LIN {X 0,Y 672.032,Z 834.911,A -85,B 0,C 180,E1 31418.47,E2 31418.47} C_VEL
LIN {X 0,Y 671.95,Z 841.394,A -85,B 0,C 180,E1 31416.751,E2 31416.751} C_VEL
LIN {X 0,Y 671.913,Z 846.943,A -85,B 0,C 180,E1 31414.78,E2 31414.78} C_VEL
LIN {X 0,Y 671.901,Z 850.246,A -85,B 0,C 180,E1 31412.986,E2 31412.986} C_VEL
LIN {X 0,Y 671.897,Z 851.95,A -85,B 0,C 180,E1 31411.364,E2 31411.364} C_VEL
LIN {X 0,Y 671.9,Z 852.431,A -85,B 0,C 180,E1 31409.574,E2 31409.574} C_VEL
LIN {X 0,Y 671.909,Z 851.064,A -85,B 0,C 180,E1 31407.527,E2 31407.527} C_VEL
LIN {X 0,Y 671.923,Z 848.206,A -85,B 0,C 180,E1 31405.733,E2 31405.733} C_VEL
LIN {X 0,Y 671.94,Z 844.025,A -85,B 0,C 180,E1 31404.021,E2 31404.021} C_VEL
LIN {X 0,Y 671.981,Z 838.375,A -85,B 0,C 180,E1 31402.304,E2 31402.304} C_VEL
LIN {X 0,Y 672.106,Z 829.893,A -85,B 0,C 180,E1 31400.322,E2 31400.322} C_VEL
LIN {X 0,Y 672.271,Z 821.072,A -85,B 0,C 180,E1 31398.678,E2 31398.678} C_VEL
LIN {X 0,Y 672.494,Z 811.756,A -85,B 0,C 180,E1 31397.201,E2 31397.201} C_VEL
LIN {X 0,Y 672.852,Z 799.566,A -85,B 0,C 180,E1 31395.543,E2 31395.543} C_VEL
LIN {X 0,Y 673.329,Z 784.965,A -85,B 0,C 180,E1 31393.877,E2 31393.877} C_VEL
LIN {X 0,Y 673.81,Z 771.549,A -85,B 0,C 180,E1 31392.557,E2 31392.557} C_VEL
LIN {X 0,Y 674.343,Z 757.55,A -85,B 0,C 180,E1 31391.35,E2 31391.35} C_VEL
LIN {X 0,Y 674.979,Z 741.859,A -85,B 0,C 180,E1 31390.165,E2 31390.165} C_VEL
LIN {X 0,Y 675.763,Z 721.934,A -85,B 0,C 180,E1 31388.882,E2 31388.882} C_VEL
LIN {X 0,Y 676.425,Z 704.738,A -85,B 0,C 180,E1 31387.947,E2 31387.947} C_VEL
LIN {X 0,Y 676.991,Z 688.587,A -85,B 0,C 180,E1 31387.188,E2 31387.188} C_VEL
LIN {X 0,Y 677.555,Z 671.856,A -85,B 0,C 180,E1 31386.519,E2 31386.519} C_VEL
LIN {X 0,Y 678.053,Z 655.221,A -85,B 0,C 180,E1 31385.96,E2 31385.96} C_VEL
LIN {X 0,Y 678.51,Z 638.285,A -85,B 0,C 180,E1 31385.494,E2 31385.494} C_VEL
LIN {X 0,Y 678.88,Z 621.075,A -85,B 0,C 180,E1 31385.12,E2 31385.12} C_VEL
LIN {X 0,Y 679.16,Z 603.568,A -85,B 0,C 180,E1 31384.84,E2 31384.84} C_VEL
LIN {X 0,Y 681.182,Z 326.681,A -85,B 0,C 180,E1 31381.687,E2 31381.687} C_VEL
LIN {X 0,Y 681.006,Z 317.975,A -85,B 0,C 180,E1 31381.575,E2 31381.575} C_VEL
LIN {X 0,Y 679.405,Z 309.493,A -85,B 0,C 180,E1 31381.377,E2 31381.377} C_VEL
LIN {X 0,Y 680.471,Z 276.701,A -85,B 0,C 180,E1 31379.001,E2 31379.001} C_VEL
LIN {X 0,Y 681.79,Z 234.937,A -85,B 0,C 180,E1 31375.957,E2 31375.957} C_VEL
LIN {X 0,Y 681.872,Z 225.908,A -85,B 0,C 180,E1 31375.284,E2 31375.284} C_VEL
LIN {X 0,Y 675.939,Z 210.334,A -85,B 0,C 180,E1 31373.798,E2 31373.798} C_VEL
LIN {X 0,Y 672.552,Z 201.457,A -85,B 0,C 180,E1 31372.978,E2 31372.978} C_VEL
LIN {X 0,Y 672.581,Z 201.453,A -85,B 0,C 180,E1 31370.042,E2 31370.042} C_VEL
LIN {X 0,Y 672.558,Z 201.452,A -85,B 0,C 180,E1 31367.085,E2 31367.085} C_VEL
LIN {X 0,Y 672.581,Z 201.448,A -85,B 0,C 180,E1 31364.087,E2 31364.087} C_VEL
LIN {X 0,Y 672.561,Z 201.45,A -85,B 0,C 180,E1 31361.081,E2 31361.081} C_VEL
LIN {X 0,Y 672.58,Z 201.45,A -85,B 0,C 180,E1 31358.095,E2 31358.095} C_VEL
LIN {X 0,Y 672.565,Z 201.448,A -85,B 0,C 180,E1 31355.02,E2 31355.02} C_VEL
LIN {X 0,Y 672.578,Z 201.451,A -85,B 0,C 180,E1 31352.055,E2 31352.055} C_VEL
LIN {X 0,Y 672.57,Z 201.443,A -85,B 0,C 180,E1 31349.054,E2 31349.054} C_VEL
LIN {X 0,Y 672.575,Z 201.452,A -85,B 0,C 180,E1 31346.013,E2 31346.013} C_VEL
LIN {X 0,Y 672.573,Z 201.435,A -85,B 0,C 180,E1 31343.016,E2 31343.016} C_VEL
LIN {X 0,Y 672.572,Z 201.448,A -85,B 0,C 180,E1 31339.995,E2 31339.995} C_VEL
LIN {X 0,Y 672.574,Z 201.438,A -85,B 0,C 180,E1 31336.941,E2 31336.941} C_VEL
LIN {X 0,Y 672.569,Z 201.445,A -85,B 0,C 180,E1 31333.936,E2 31333.936} C_VEL
LIN {X 0,Y 672.576,Z 201.439,A -85,B 0,C 180,E1 31330.883,E2 31330.883} C_VEL
LIN {X 0,Y 672.565,Z 201.446,A -85,B 0,C 180,E1 31327.861,E2 31327.861} C_VEL
LIN {X 0,Y 672.579,Z 201.437,A -85,B 0,C 180,E1 31324.861,E2 31324.861} C_VEL
LIN {X 0,Y 672.561,Z 201.448,A -85,B 0,C 180,E1 31321.789,E2 31321.789} C_VEL
LIN {X 0,Y 672.581,Z 201.432,A -85,B 0,C 180,E1 31318.807,E2 31318.807} C_VEL
LIN {X 0,Y 672.557,Z 201.451,A -85,B 0,C 180,E1 31315.737,E2 31315.737} C_VEL
LIN {X 0,Y 672.582,Z 201.433,A -85,B 0,C 180,E1 31312.74,E2 31312.74} C_VEL
LIN {X 0,Y 672.555,Z 201.452,A -85,B 0,C 180,E1 31309.723,E2 31309.723} C_VEL
LIN {X 0,Y 672.586,Z 201.445,A -85,B 0,C 180,E1 31306.765,E2 31306.765} C_VEL
LIN {X 0,Y 672.554,Z 201.454,A -85,B 0,C 180,E1 31303.77,E2 31303.77} C_VEL
LIN {X 0,Y 672.582,Z 201.444,A -85,B 0,C 180,E1 31300.819,E2 31300.819} C_VEL
LIN {X 0,Y 672.552,Z 201.454,A -85,B 0,C 180,E1 31297.721,E2 31297.721} C_VEL
LIN {X 0,Y 672.581,Z 201.446,A -85,B 0,C 180,E1 31294.744,E2 31294.744} C_VEL
LIN {X 0,Y 672.547,Z 201.453,A -85,B 0,C 180,E1 31291.659,E2 31291.659} C_VEL
LIN {X 0,Y 672.578,Z 201.447,A -85,B 0,C 180,E1 31288.74,E2 31288.74} C_VEL
LIN {X 0,Y 672.549,Z 201.455,A -85,B 0,C 180,E1 31285.704,E2 31285.704} C_VEL
LIN {X 0,Y 672.559,Z 201.449,A -85,B 0,C 180,E1 31282.832,E2 31282.832} C_VEL
LIN {X 0,Y 672.548,Z 201.456,A -85,B 0,C 180,E1 31279.702,E2 31279.702} C_VEL
LIN {X 0,Y 672.55,Z 201.452,A -85,B 0,C 180,E1 31276.851,E2 31276.851} C_VEL
LIN {X 0,Y 672.552,Z 201.458,A -85,B 0,C 180,E1 31273.735,E2 31273.735} C_VEL
LIN {X 0,Y 672.57,Z 201.682,A -85,B 0,C 180,E1 31272.914,E2 31272.914} C_VEL
LIN {X 0,Y 673.919,Z 205.007,A -85,B 0,C 180,E1 31272.615,E2 31272.615} C_VEL
LIN {X 0,Y 682.61,Z 222.727,A -85,B 0,C 180,E1 31270.965,E2 31270.965} C_VEL
LIN {X 0,Y 686.788,Z 232.051,A -85,B 0,C 180,E1 31270.19,E2 31270.19} C_VEL
LIN {X 0,Y 684.973,Z 290.804,A -85,B 0,C 180,E1 31267.339,E2 31267.339} C_VEL
LIN {X 0,Y 684.73,Z 300.754,A -85,B 0,C 180,E1 31266.874,E2 31266.874} C_VEL
LIN {X 0,Y 686.841,Z 315.173,A -85,B 0,C 180,E1 31266.576,E2 31266.576} C_VEL
LIN {X 0,Y 685.386,Z 510.12,A -85,B 0,C 180,E1 31264.28,E2 31264.28} C_VEL
LIN {X 0,Y 683.704,Z 691.141,A -85,B 0,C 180,E1 31262.122,E2 31262.122} C_VEL
LIN {X 0,Y 683.128,Z 716.495,A -85,B 0,C 180,E1 31261.672,E2 31261.672} C_VEL
LIN {X 0,Y 682.438,Z 738.1,A -85,B 0,C 180,E1 31261.152,E2 31261.152} C_VEL
LIN {X 0,Y 681.652,Z 761.266,A -85,B 0,C 180,E1 31260.451,E2 31260.451} C_VEL
LIN {X 0,Y 680.761,Z 782.216,A -85,B 0,C 180,E1 31259.668,E2 31259.668} C_VEL
LIN {X 0,Y 679.885,Z 802.279,A -85,B 0,C 180,E1 31258.793,E2 31258.793} C_VEL
LIN {X 0,Y 678.731,Z 825.506,A -85,B 0,C 180,E1 31257.601,E2 31257.601} C_VEL
LIN {X 0,Y 677.787,Z 844.732,A -85,B 0,C 180,E1 31256.457,E2 31256.457} C_VEL
LIN {X 0,Y 676.663,Z 866.009,A -85,B 0,C 180,E1 31255,E2 31255} C_VEL
LIN {X 0,Y 675.802,Z 883.401,A -85,B 0,C 180,E1 31253.638,E2 31253.638} C_VEL
LIN {X 0,Y 674.846,Z 902.606,A -85,B 0,C 180,E1 31251.924,E2 31251.924} C_VEL
LIN {X 0,Y 674.159,Z 917.749,A -85,B 0,C 180,E1 31250.386,E2 31250.386} C_VEL
LIN {X 0,Y 673.471,Z 933.816,A -85,B 0,C 180,E1 31248.525,E2 31248.525} C_VEL
LIN {X 0,Y 673.017,Z 946.526,A -85,B 0,C 180,E1 31246.84,E2 31246.84} C_VEL
LIN {X 0,Y 672.589,Z 959.764,A -85,B 0,C 180,E1 31244.815,E2 31244.815} C_VEL
LIN {X 0,Y 672.315,Z 969.606,A -85,B 0,C 180,E1 31243.058,E2 31243.058} C_VEL
LIN {X 0,Y 672.101,Z 979.477,A -85,B 0,C 180,E1 31240.978,E2 31240.978} C_VEL
LIN {X 0,Y 672.004,Z 986.514,A -85,B 0,C 180,E1 31239.161,E2 31239.161} C_VEL
LIN {X 0,Y 671.934,Z 992.507,A -85,B 0,C 180,E1 31237.267,E2 31237.267} C_VEL
LIN {X 0,Y 671.893,Z 997.337,A -85,B 0,C 180,E1 31235.208,E2 31235.208} C_VEL
LIN {X 0,Y 671.908,Z 1000.237,A -85,B 0,C 180,E1 31233.413,E2 31233.413} C_VEL
LIN {X 0,Y 671.908,Z 1002.17,A -85,B 0,C 180,E1 31231.279,E2 31231.279} C_VEL
LIN {X 0,Y 671.882,Z 1002.351,A -85,B 0,C 180,E1 31229.403,E2 31229.403} C_VEL
LIN {X 0,Y 671.907,Z 1001.363,A -85,B 0,C 180,E1 31227.612,E2 31227.612} C_VEL
LIN {X 0,Y 671.918,Z 998.608,A -85,B 0,C 180,E1 31225.476,E2 31225.476} C_VEL
LIN {X 0,Y 671.925,Z 994.689,A -85,B 0,C 180,E1 31223.592,E2 31223.592} C_VEL
LIN {X 0,Y 671.975,Z 989.201,A -85,B 0,C 180,E1 31221.615,E2 31221.615} C_VEL
LIN {X 0,Y 672.091,Z 981.605,A -85,B 0,C 180,E1 31219.543,E2 31219.543} C_VEL
LIN {X 0,Y 672.253,Z 973.118,A -85,B 0,C 180,E1 31217.632,E2 31217.632} C_VEL
LIN {X 0,Y 672.515,Z 962.354,A -85,B 0,C 180,E1 31215.623,E2 31215.623} C_VEL
LIN {X 0,Y 672.843,Z 951.388,A -85,B 0,C 180,E1 31213.865,E2 31213.865} C_VEL
LIN {X 0,Y 673.361,Z 936.945,A -85,B 0,C 180,E1 31211.871,E2 31211.871} C_VEL
LIN {X 0,Y 673.931,Z 922.728,A -85,B 0,C 180,E1 31210.161,E2 31210.161} C_VEL
LIN {X 0,Y 674.685,Z 906.31,A -85,B 0,C 180,E1 31208.436,E2 31208.436} C_VEL
LIN {X 0,Y 675.451,Z 890.139,A -85,B 0,C 180,E1 31206.935,E2 31206.935} C_VEL
LIN {X 0,Y 676.436,Z 870.867,A -85,B 0,C 180,E1 31205.364,E2 31205.364} C_VEL
LIN {X 0,Y 677.326,Z 853.071,A -85,B 0,C 180,E1 31204.09,E2 31204.09} C_VEL
LIN {X 0,Y 678.489,Z 830.879,A -85,B 0,C 180,E1 31202.704,E2 31202.704} C_VEL
LIN {X 0,Y 679.431,Z 811.337,A -85,B 0,C 180,E1 31201.649,E2 31201.649} C_VEL
LIN {X 0,Y 680.53,Z 787.863,A -85,B 0,C 180,E1 31200.562,E2 31200.562} C_VEL
LIN {X 0,Y 681.37,Z 767.685,A -85,B 0,C 180,E1 31199.778,E2 31199.778} C_VEL
LIN {X 0,Y 682.256,Z 745.15,A -85,B 0,C 180,E1 31199.042,E2 31199.042} C_VEL
LIN {X 0,Y 682.957,Z 721.163,A -85,B 0,C 180,E1 31198.429,E2 31198.429} C_VEL
LIN {X 0,Y 683.574,Z 698.388,A -85,B 0,C 180,E1 31197.987,E2 31197.987} C_VEL
LIN {X 0,Y 684.015,Z 664.777,A -85,B 0,C 180,E1 31197.547,E2 31197.547} C_VEL
LIN {X 0,Y 686.084,Z 426.859,A -85,B 0,C 180,E1 31194.728,E2 31194.728} C_VEL
LIN {X 0,Y 686.203,Z 312.509,A -85,B 0,C 180,E1 31193.45,E2 31193.45} C_VEL
LIN {X 0,Y 684.133,Z 300.68,A -85,B 0,C 180,E1 31193.219,E2 31193.219} C_VEL
LIN {X 0,Y 685,Z 265.459,A -85,B 0,C 180,E1 31191.55,E2 31191.55} C_VEL
LIN {X 0,Y 686.519,Z 233.708,A -85,B 0,C 180,E1 31189.927,E2 31189.927} C_VEL
LIN {X 0,Y 686.523,Z 231.357,A -85,B 0,C 180,E1 31189.791,E2 31189.791} C_VEL
LIN {X 0,Y 680.861,Z 218.547,A -85,B 0,C 180,E1 31188.502,E2 31188.502} C_VEL
LIN {X 0,Y 676.932,Z 210.351,A -85,B 0,C 180,E1 31187.483,E2 31187.483} C_VEL
LIN {X 0,Y 674.606,Z 205.849,A -85,B 0,C 180,E1 31186.823,E2 31186.823} C_VEL
LIN {X 0,Y 672.75,Z 202.49,A -85,B 0,C 180,E1 31186.247,E2 31186.247} C_VEL
LIN {X 0,Y 672.552,Z 201.458,A -85,B 0,C 180,E1 31186.094,E2 31186.094} C_VEL
LIN {X 0,Y 672.565,Z 201.456,A -85,B 0,C 180,E1 31182.914,E2 31182.914} C_VEL
LIN {X 0,Y 672.538,Z 201.46,A -85,B 0,C 180,E1 31180.073,E2 31180.073} C_VEL
LIN {X 0,Y 672.614,Z 201.669,A -85,B 0,C 180,E1 31177.633,E2 31177.633} C_VEL
LIN {X 0,Y 674.124,Z 205.273,A -85,B 0,C 180,E1 31177.062,E2 31177.062} C_VEL
LIN {X 0,Y 675.014,Z 206.813,A -85,B 0,C 180,E1 31176.809,E2 31176.809} C_VEL
LIN {X 0,Y 678.723,Z 215.05,A -85,B 0,C 180,E1 31175.689,E2 31175.689} C_VEL
LIN {X 0,Y 683.33,Z 226.73,A -85,B 0,C 180,E1 31174.383,E2 31174.383} C_VEL
LIN {X 0,Y 683.402,Z 229.375,A -85,B 0,C 180,E1 31174.183,E2 31174.183} C_VEL
LIN {X 0,Y 680.701,Z 272.496,A -85,B 0,C 180,E1 31171.412,E2 31171.412} C_VEL
LIN {X 0,Y 678.57,Z 326.363,A -85,B 0,C 180,E1 31168.134,E2 31168.134} C_VEL
LIN {X 0,Y 677.146,Z 378.659,A -85,B 0,C 180,E1 31165.074,E2 31165.074} C_VEL
LIN {X 0,Y 675.934,Z 433.54,A -85,B 0,C 180,E1 31161.951,E2 31161.951} C_VEL
LIN {X 0,Y 675.545,Z 457.444,A -85,B 0,C 180,E1 31160.632,E2 31160.632} C_VEL
LIN {X 0,Y 678.294,Z 481.315,A -85,B 0,C 180,E1 31160.165,E2 31160.165} C_VEL
LIN {X 0,Y 676.325,Z 608.391,A -85,B 0,C 180,E1 31158.536,E2 31158.536} C_VEL
LIN {X 0,Y 675.634,Z 682.185,A -85,B 0,C 180,E1 31157.622,E2 31157.622} C_VEL
LIN {X 0,Y 675.344,Z 701.727,A -85,B 0,C 180,E1 31157.222,E2 31157.222} C_VEL
LIN {X 0,Y 675.02,Z 719.823,A -85,B 0,C 180,E1 31156.7,E2 31156.7} C_VEL
LIN {X 0,Y 674.636,Z 737.26,A -85,B 0,C 180,E1 31156.046,E2 31156.046} C_VEL
LIN {X 0,Y 674.245,Z 754.12,A -85,B 0,C 180,E1 31155.251,E2 31155.251} C_VEL
LIN {X 0,Y 673.837,Z 770.294,A -85,B 0,C 180,E1 31154.31,E2 31154.31} C_VEL
LIN {X 0,Y 673.428,Z 785.113,A -85,B 0,C 180,E1 31153.262,E2 31153.262} C_VEL
LIN {X 0,Y 673.048,Z 798.81,A -85,B 0,C 180,E1 31152.091,E2 31152.091} C_VEL
LIN {X 0,Y 672.736,Z 810.592,A -85,B 0,C 180,E1 31150.881,E2 31150.881} C_VEL
LIN {X 0,Y 672.473,Z 821.059,A -85,B 0,C 180,E1 31149.586,E2 31149.586} C_VEL
LIN {X 0,Y 672.265,Z 830.19,A -85,B 0,C 180,E1 31148.209,E2 31148.209} C_VEL
LIN {X 0,Y 672.124,Z 837.938,A -85,B 0,C 180,E1 31146.749,E2 31146.749} C_VEL
LIN {X 0,Y 672.045,Z 844.23,A -85,B 0,C 180,E1 31145.207,E2 31145.207} C_VEL
LIN {X 0,Y 671.982,Z 848.97,A -85,B 0,C 180,E1 31143.583,E2 31143.583} C_VEL
LIN {X 0,Y 671.955,Z 852.015,A -85,B 0,C 180,E1 31141.876,E2 31141.876} C_VEL
LIN {X 0,Y 671.948,Z 853.148,A -85,B 0,C 180,E1 31140.256,E2 31140.256} C_VEL
LIN {X 0,Y 671.945,Z 852.596,A -85,B 0,C 180,E1 31138.636,E2 31138.636} C_VEL
LIN {X 0,Y 671.96,Z 850.344,A -85,B 0,C 180,E1 31137.015,E2 31137.015} C_VEL
LIN {X 0,Y 671.989,Z 846.324,A -85,B 0,C 180,E1 31135.391,E2 31135.391} C_VEL
LIN {X 0,Y 672.056,Z 840.398,A -85,B 0,C 180,E1 31133.765,E2 31133.765} C_VEL
LIN {X 0,Y 672.168,Z 832.667,A -85,B 0,C 180,E1 31132.187,E2 31132.187} C_VEL
LIN {X 0,Y 672.345,Z 823.743,A -85,B 0,C 180,E1 31130.757,E2 31130.757} C_VEL
LIN {X 0,Y 672.591,Z 813.122,A -85,B 0,C 180,E1 31129.377,E2 31129.377} C_VEL
LIN {X 0,Y 672.898,Z 800.975,A -85,B 0,C 180,E1 31128.08,E2 31128.08} C_VEL
LIN {X 0,Y 673.268,Z 787.237,A -85,B 0,C 180,E1 31126.866,E2 31126.866} C_VEL
LIN {X 0,Y 673.678,Z 772.328,A -85,B 0,C 180,E1 31125.776,E2 31125.776} C_VEL
LIN {X 0,Y 674.102,Z 756.538,A -85,B 0,C 180,E1 31124.823,E2 31124.823} C_VEL
LIN {X 0,Y 674.498,Z 739.713,A -85,B 0,C 180,E1 31123.994,E2 31123.994} C_VEL
LIN {X 0,Y 674.919,Z 721.886,A -85,B 0,C 180,E1 31123.297,E2 31123.297} C_VEL
LIN {X 0,Y 675.274,Z 702.619,A -85,B 0,C 180,E1 31122.724,E2 31122.724} C_VEL
LIN {X 0,Y 675.562,Z 683.284,A -85,B 0,C 180,E1 31122.32,E2 31122.32} C_VEL
LIN {X 0,Y 675.824,Z 651.623,A -85,B 0,C 180,E1 31121.921,E2 31121.921} C_VEL
LIN {X 0,Y 676.454,Z 561.656,A -85,B 0,C 180,E1 31120.895,E2 31120.895} C_VEL
LIN {X 0,Y 675.607,Z 554.064,A -85,B 0,C 180,E1 31120.777,E2 31120.777} C_VEL
LIN {X 0,Y 669.963,Z 534.195,A -85,B 0,C 180,E1 31120.351,E2 31120.351} C_VEL
LIN {X 0,Y 669.337,Z 527.67,A -85,B 0,C 180,E1 31120.25,E2 31120.25} C_VEL
LIN {X 0,Y 669.559,Z 478.594,A -85,B 0,C 180,E1 31119.656,E2 31119.656} C_VEL
LIN {X 0,Y 667.897,Z 464.609,A -85,B 0,C 180,E1 31119.402,E2 31119.402} C_VEL
LIN {X 0,Y 669.123,Z 409.096,A -85,B 0,C 180,E1 31116.251,E2 31116.251} C_VEL
LIN {X 0,Y 670.415,Z 355.832,A -85,B 0,C 180,E1 31113.181,E2 31113.181} C_VEL
LIN {X 0,Y 671.812,Z 303.955,A -85,B 0,C 180,E1 31110.142,E2 31110.142} C_VEL
LIN {X 0,Y 673.338,Z 252.657,A -85,B 0,C 180,E1 31107.078,E2 31107.078} C_VEL
LIN {X 0,Y 674.106,Z 227.628,A -85,B 0,C 180,E1 31105.559,E2 31105.559} C_VEL
LIN {X 0,Y 664.614,Z 202.433,A -85,B 0,C 180,E1 31103.405,E2 31103.405} C_VEL
LIN {X 0,Y 664.637,Z 202.442,A -85,B 0,C 180,E1 31100.366,E2 31100.366} C_VEL
LIN {X 0,Y 664.598,Z 202.446,A -85,B 0,C 180,E1 31097.494,E2 31097.494} C_VEL
LIN {X 0,Y 664.644,Z 202.437,A -85,B 0,C 180,E1 31094.39,E2 31094.39} C_VEL
LIN {X 0,Y 664.607,Z 202.442,A -85,B 0,C 180,E1 31091.336,E2 31091.336} C_VEL
LIN {X 0,Y 664.64,Z 202.444,A -85,B 0,C 180,E1 31088.39,E2 31088.39} C_VEL
LIN {X 0,Y 664.587,Z 202.509,A -85,B 0,C 180,E1 31087.338,E2 31087.338} C_VEL
LIN {X 0,Y 667.131,Z 208.973,A -85,B 0,C 180,E1 31086.764,E2 31086.764} C_VEL
LIN {X 0,Y 673.998,Z 226.544,A -85,B 0,C 180,E1 31085.098,E2 31085.098} C_VEL
LIN {X 0,Y 675.119,Z 230.081,A -85,B 0,C 180,E1 31084.765,E2 31084.765} C_VEL
LIN {X 0,Y 673.763,Z 269.836,A -85,B 0,C 180,E1 31081.842,E2 31081.842} C_VEL
LIN {X 0,Y 672.675,Z 312.651,A -85,B 0,C 180,E1 31078.795,E2 31078.795} C_VEL
LIN {X 0,Y 674.226,Z 321.813,A -85,B 0,C 180,E1 31078.608,E2 31078.608} C_VEL
LIN {X 0,Y 672.018,Z 576.504,A -85,B 0,C 180,E1 31075.653,E2 31075.653} C_VEL
LIN {X 0,Y 671.7,Z 612.862,A -85,B 0,C 180,E1 31075.21,E2 31075.21} C_VEL
LIN {X 0,Y 671.233,Z 635.63,A -85,B 0,C 180,E1 31074.757,E2 31074.757} C_VEL
LIN {X 0,Y 670.779,Z 653.07,A -85,B 0,C 180,E1 31074.294,E2 31074.294} C_VEL
LIN {X 0,Y 670.25,Z 669.467,A -85,B 0,C 180,E1 31073.753,E2 31073.753} C_VEL
LIN {X 0,Y 669.63,Z 686.01,A -85,B 0,C 180,E1 31073.101,E2 31073.101} C_VEL
LIN {X 0,Y 669.013,Z 702.077,A -85,B 0,C 180,E1 31072.357,E2 31072.357} C_VEL
LIN {X 0,Y 668.387,Z 717.241,A -85,B 0,C 180,E1 31071.547,E2 31071.547} C_VEL
LIN {X 0,Y 667.726,Z 732.366,A -85,B 0,C 180,E1 31070.624,E2 31070.624} C_VEL
LIN {X 0,Y 667.085,Z 746.814,A -85,B 0,C 180,E1 31069.618,E2 31069.618} C_VEL
LIN {X 0,Y 666.436,Z 762.21,A -85,B 0,C 180,E1 31068.398,E2 31068.398} C_VEL
LIN {X 0,Y 665.739,Z 778.959,A -85,B 0,C 180,E1 31066.85,E2 31066.85} C_VEL
LIN {X 0,Y 665.22,Z 792.126,A -85,B 0,C 180,E1 31065.429,E2 31065.429} C_VEL
LIN {X 0,Y 664.825,Z 803.575,A -85,B 0,C 180,E1 31064.013,E2 31064.013} C_VEL
LIN {X 0,Y 664.513,Z 814.084,A -85,B 0,C 180,E1 31062.514,E2 31062.514} C_VEL
LIN {X 0,Y 664.233,Z 825.477,A -85,B 0,C 180,E1 31060.583,E2 31060.583} C_VEL
LIN {X 0,Y 664.065,Z 833.798,A -85,B 0,C 180,E1 31058.835,E2 31058.835} C_VEL
LIN {X 0,Y 663.983,Z 839.878,A -85,B 0,C 180,E1 31057.267,E2 31057.267} C_VEL
LIN {X 0,Y 663.933,Z 844.97,A -85,B 0,C 180,E1 31055.618,E2 31055.618} C_VEL
LIN {X 0,Y 663.918,Z 849.209,A -85,B 0,C 180,E1 31053.713,E2 31053.713} C_VEL
LIN {X 0,Y 663.913,Z 851.709,A -85,B 0,C 180,E1 31051.726,E2 31051.726} C_VEL
LIN {X 0,Y 663.919,Z 852.424,A -85,B 0,C 180,E1 31050,E2 31050} C_VEL
LIN {X 0,Y 663.911,Z 851.771,A -85,B 0,C 180,E1 31048.274,E2 31048.274} C_VEL
LIN {X 0,Y 663.917,Z 849.529,A -85,B 0,C 180,E1 31046.373,E2 31046.373} C_VEL
LIN {X 0,Y 663.936,Z 845.22,A -85,B 0,C 180,E1 31044.382,E2 31044.382} C_VEL
LIN {X 0,Y 663.98,Z 840.192,A -85,B 0,C 180,E1 31042.733,E2 31042.733} C_VEL
LIN {X 0,Y 664.054,Z 834.18,A -85,B 0,C 180,E1 31041.165,E2 31041.165} C_VEL
LIN {X 0,Y 664.223,Z 825.939,A -85,B 0,C 180,E1 31039.417,E2 31039.417} C_VEL
LIN {X 0,Y 664.494,Z 814.683,A -85,B 0,C 180,E1 31037.486,E2 31037.486} C_VEL
LIN {X 0,Y 664.807,Z 804.016,A -85,B 0,C 180,E1 31035.955,E2 31035.955} C_VEL
LIN {X 0,Y 665.191,Z 792.891,A -85,B 0,C 180,E1 31034.57,E2 31034.57} C_VEL
LIN {X 0,Y 665.655,Z 780.673,A -85,B 0,C 180,E1 31033.237,E2 31033.237} C_VEL
LIN {X 0,Y 666.33,Z 764.724,A -85,B 0,C 180,E1 31031.722,E2 31031.722} C_VEL
LIN {X 0,Y 667.041,Z 748.021,A -85,B 0,C 180,E1 31030.38,E2 31030.38} C_VEL
LIN {X 0,Y 667.68,Z 733.331,A -85,B 0,C 180,E1 31029.349,E2 31029.349} C_VEL
LIN {X 0,Y 668.355,Z 717.99,A -85,B 0,C 180,E1 31028.406,E2 31028.406} C_VEL
LIN {X 0,Y 668.982,Z 702.926,A -85,B 0,C 180,E1 31027.596,E2 31027.596} C_VEL
LIN {X 0,Y 669.569,Z 687.517,A -85,B 0,C 180,E1 31026.875,E2 31026.875} C_VEL
LIN {X 0,Y 670.158,Z 671.819,A -85,B 0,C 180,E1 31026.244,E2 31026.244} C_VEL
LIN {X 0,Y 670.68,Z 655.903,A -85,B 0,C 180,E1 31025.702,E2 31025.702} C_VEL
LIN {X 0,Y 671.137,Z 639.382,A -85,B 0,C 180,E1 31025.245,E2 31025.245} C_VEL
LIN {X 0,Y 671.516,Z 621.739,A -85,B 0,C 180,E1 31024.861,E2 31024.861} C_VEL
LIN {X 0,Y 671.791,Z 603.592,A -85,B 0,C 180,E1 31024.573,E2 31024.573} C_VEL
LIN {X 0,Y 673.859,Z 361.059,A -85,B 0,C 180,E1 31021.758,E2 31021.758} C_VEL
LIN {X 0,Y 674.06,Z 319.616,A -85,B 0,C 180,E1 31021.265,E2 31021.265} C_VEL
LIN {X 0,Y 672.599,Z 311.902,A -85,B 0,C 180,E1 31021.085,E2 31021.085} C_VEL
LIN {X 0,Y 673.656,Z 272.529,A -85,B 0,C 180,E1 31018.265,E2 31018.265} C_VEL
LIN {X 0,Y 675.029,Z 233.352,A -85,B 0,C 180,E1 31015.385,E2 31015.385} C_VEL
LIN {X 0,Y 674.99,Z 229.369,A -85,B 0,C 180,E1 31015.085,E2 31015.085} C_VEL
LIN {X 0,Y 668.438,Z 212.229,A -85,B 0,C 180,E1 31013.445,E2 31013.445} C_VEL
LIN {X 0,Y 664.641,Z 202.534,A -85,B 0,C 180,E1 31012.571,E2 31012.571} C_VEL
LIN {X 0,Y 664.632,Z 202.437,A -85,B 0,C 180,E1 31009.352,E2 31009.352} C_VEL
LIN {X 0,Y 664.643,Z 202.438,A -85,B 0,C 180,E1 31006.329,E2 31006.329} C_VEL
LIN {X 0,Y 664.627,Z 202.434,A -85,B 0,C 180,E1 31003.198,E2 31003.198} C_VEL
LIN {X 0,Y 664.645,Z 202.437,A -85,B 0,C 180,E1 31000.161,E2 31000.161} C_VEL
LIN {X 0,Y 664.628,Z 202.433,A -85,B 0,C 180,E1 30997.105,E2 30997.105} C_VEL
LIN {X 0,Y 664.637,Z 202.436,A -85,B 0,C 180,E1 30994.031,E2 30994.031} C_VEL
LIN {X 0,Y 664.626,Z 202.437,A -85,B 0,C 180,E1 30990.96,E2 30990.96} C_VEL
LIN {X 0,Y 664.636,Z 202.435,A -85,B 0,C 180,E1 30987.982,E2 30987.982} C_VEL
LIN {X 0,Y 664.629,Z 202.436,A -85,B 0,C 180,E1 30984.913,E2 30984.913} C_VEL
LIN {X 0,Y 664.633,Z 202.439,A -85,B 0,C 180,E1 30981.907,E2 30981.907} C_VEL
LIN {X 0,Y 664.632,Z 202.431,A -85,B 0,C 180,E1 30978.865,E2 30978.865} C_VEL
LIN {X 0,Y 664.63,Z 202.44,A -85,B 0,C 180,E1 30975.891,E2 30975.891} C_VEL
LIN {X 0,Y 664.635,Z 202.428,A -85,B 0,C 180,E1 30972.865,E2 30972.865} C_VEL
LIN {X 0,Y 664.625,Z 202.44,A -85,B 0,C 180,E1 30969.788,E2 30969.788} C_VEL
LIN {X 0,Y 664.636,Z 202.431,A -85,B 0,C 180,E1 30966.739,E2 30966.739} C_VEL
LIN {X 0,Y 664.621,Z 202.439,A -85,B 0,C 180,E1 30963.709,E2 30963.709} C_VEL
LIN {X 0,Y 664.637,Z 202.434,A -85,B 0,C 180,E1 30960.69,E2 30960.69} C_VEL
LIN {X 0,Y 664.616,Z 202.438,A -85,B 0,C 180,E1 30957.672,E2 30957.672} C_VEL
LIN {X 0,Y 664.641,Z 202.436,A -85,B 0,C 180,E1 30954.648,E2 30954.648} C_VEL
LIN {X 0,Y 664.615,Z 202.437,A -85,B 0,C 180,E1 30951.696,E2 30951.696} C_VEL
LIN {X 0,Y 664.645,Z 202.435,A -85,B 0,C 180,E1 30948.722,E2 30948.722} C_VEL
LIN {X 0,Y 664.613,Z 202.439,A -85,B 0,C 180,E1 30945.668,E2 30945.668} C_VEL
LIN {X 0,Y 664.647,Z 202.436,A -85,B 0,C 180,E1 30942.67,E2 30942.67} C_VEL
LIN {X 0,Y 664.608,Z 202.44,A -85,B 0,C 180,E1 30939.602,E2 30939.602} C_VEL
LIN {X 0,Y 664.649,Z 202.437,A -85,B 0,C 180,E1 30936.589,E2 30936.589} C_VEL
LIN {X 0,Y 664.604,Z 202.438,A -85,B 0,C 180,E1 30933.53,E2 30933.53} C_VEL
LIN {X 0,Y 664.65,Z 202.436,A -85,B 0,C 180,E1 30930.532,E2 30930.532} C_VEL
LIN {X 0,Y 664.601,Z 202.443,A -85,B 0,C 180,E1 30927.513,E2 30927.513} C_VEL
LIN {X 0,Y 664.643,Z 202.438,A -85,B 0,C 180,E1 30924.606,E2 30924.606} C_VEL
LIN {X 0,Y 664.601,Z 202.444,A -85,B 0,C 180,E1 30921.584,E2 30921.584} C_VEL
LIN {X 0,Y 664.633,Z 202.439,A -85,B 0,C 180,E1 30918.666,E2 30918.666} C_VEL
LIN {X 0,Y 664.601,Z 202.446,A -85,B 0,C 180,E1 30915.606,E2 30915.606} C_VEL
LIN {X 0,Y 664.612,Z 202.564,A -85,B 0,C 180,E1 30913.505,E2 30913.505} C_VEL
LIN {X 0,Y 665.771,Z 205.742,A -85,B 0,C 180,E1 30913.223,E2 30913.223} C_VEL
LIN {X 0,Y 667.227,Z 208.56,A -85,B 0,C 180,E1 30912.941,E2 30912.941} C_VEL
LIN {X 0,Y 673.156,Z 220.579,A -85,B 0,C 180,E1 30911.784,E2 30911.784} C_VEL
LIN {X 0,Y 679.957,Z 234.951,A -85,B 0,C 180,E1 30910.513,E2 30910.513} C_VEL
LIN {X 0,Y 680.142,Z 237.631,A -85,B 0,C 180,E1 30910.36,E2 30910.36} C_VEL
LIN {X 0,Y 678.085,Z 294.371,A -85,B 0,C 180,E1 30907.571,E2 30907.571} C_VEL
LIN {X 0,Y 677.934,Z 301.386,A -85,B 0,C 180,E1 30907.246,E2 30907.246} C_VEL
LIN {X 0,Y 680.085,Z 316.369,A -85,B 0,C 180,E1 30906.926,E2 30906.926} C_VEL
LIN {X 0,Y 678.07,Z 580.867,A -85,B 0,C 180,E1 30903.814,E2 30903.814} C_VEL
LIN {X 0,Y 676.916,Z 691.712,A -85,B 0,C 180,E1 30902.475,E2 30902.475} C_VEL
LIN {X 0,Y 676.278,Z 717.014,A -85,B 0,C 180,E1 30902.018,E2 30902.018} C_VEL
LIN {X 0,Y 675.543,Z 738.337,A -85,B 0,C 180,E1 30901.499,E2 30901.499} C_VEL
LIN {X 0,Y 674.614,Z 762.547,A -85,B 0,C 180,E1 30900.754,E2 30900.754} C_VEL
LIN {X 0,Y 673.652,Z 783.343,A -85,B 0,C 180,E1 30899.964,E2 30899.964} C_VEL
LIN {X 0,Y 672.656,Z 804.171,A -85,B 0,C 180,E1 30899.039,E2 30899.039} C_VEL
LIN {X 0,Y 671.429,Z 826.314,A -85,B 0,C 180,E1 30897.879,E2 30897.879} C_VEL
LIN {X 0,Y 670.361,Z 846.189,A -85,B 0,C 180,E1 30896.677,E2 30896.677} C_VEL
LIN {X 0,Y 669.167,Z 866.614,A -85,B 0,C 180,E1 30895.252,E2 30895.252} C_VEL
LIN {X 0,Y 668.23,Z 883.681,A -85,B 0,C 180,E1 30893.899,E2 30893.899} C_VEL
LIN {X 0,Y 667.192,Z 902.606,A -85,B 0,C 180,E1 30892.189,E2 30892.189} C_VEL
LIN {X 0,Y 666.423,Z 917.633,A -85,B 0,C 180,E1 30890.646,E2 30890.646} C_VEL
LIN {X 0,Y 665.657,Z 933.818,A -85,B 0,C 180,E1 30888.751,E2 30888.751} C_VEL
LIN {X 0,Y 665.151,Z 946.527,A -85,B 0,C 180,E1 30887.045,E2 30887.045} C_VEL
LIN {X 0,Y 664.668,Z 959.765,A -85,B 0,C 180,E1 30884.996,E2 30884.996} C_VEL
LIN {X 0,Y 664.363,Z 969.565,A -85,B 0,C 180,E1 30883.224,E2 30883.224} C_VEL
LIN {X 0,Y 664.133,Z 979.122,A -85,B 0,C 180,E1 30881.199,E2 30881.199} C_VEL
LIN {X 0,Y 664.025,Z 986.514,A -85,B 0,C 180,E1 30879.272,E2 30879.272} C_VEL
LIN {X 0,Y 663.938,Z 992.761,A -85,B 0,C 180,E1 30877.268,E2 30877.268} C_VEL
LIN {X 0,Y 663.894,Z 997.496,A -85,B 0,C 180,E1 30875.185,E2 30875.185} C_VEL
LIN {X 0,Y 663.905,Z 1000.35,A -85,B 0,C 180,E1 30873.367,E2 30873.367} C_VEL
LIN {X 0,Y 663.911,Z 1002.193,A -85,B 0,C 180,E1 30871.208,E2 30871.208} C_VEL
LIN {X 0,Y 663.884,Z 1002.328,A -85,B 0,C 180,E1 30869.31,E2 30869.31} C_VEL
LIN {X 0,Y 663.891,Z 1001.226,A -85,B 0,C 180,E1 30867.41,E2 30867.41} C_VEL
LIN {X 0,Y 663.91,Z 998.291,A -85,B 0,C 180,E1 30865.248,E2 30865.248} C_VEL
LIN {X 0,Y 663.93,Z 994.483,A -85,B 0,C 180,E1 30863.428,E2 30863.428} C_VEL
LIN {X 0,Y 663.978,Z 988.634,A -85,B 0,C 180,E1 30861.339,E2 30861.339} C_VEL
LIN {X 0,Y 664.107,Z 981.604,A -85,B 0,C 180,E1 30859.415,E2 30859.415} C_VEL
LIN {X 0,Y 664.295,Z 973.119,A -85,B 0,C 180,E1 30857.482,E2 30857.482} C_VEL
LIN {X 0,Y 664.592,Z 962.352,A -85,B 0,C 180,E1 30855.448,E2 30855.448} C_VEL
LIN {X 0,Y 664.955,Z 951.39,A -85,B 0,C 180,E1 30853.669,E2 30853.669} C_VEL
LIN {X 0,Y 665.521,Z 937.327,A -85,B 0,C 180,E1 30851.699,E2 30851.699} C_VEL
LIN {X 0,Y 666.104,Z 924.081,A -85,B 0,C 180,E1 30850.077,E2 30850.077} C_VEL
LIN {X 0,Y 667.003,Z 906.308,A -85,B 0,C 180,E1 30848.175,E2 30848.175} C_VEL
LIN {X 0,Y 667.853,Z 890.292,A -85,B 0,C 180,E1 30846.671,E2 30846.671} C_VEL
LIN {X 0,Y 668.965,Z 870.26,A -85,B 0,C 180,E1 30845.023,E2 30845.023} C_VEL
LIN {X 0,Y 670.028,Z 851.732,A -85,B 0,C 180,E1 30843.691,E2 30843.691} C_VEL
LIN {X 0,Y 671.229,Z 830.362,A -85,B 0,C 180,E1 30842.353,E2 30842.353} C_VEL
LIN {X 0,Y 672.271,Z 810.751,A -85,B 0,C 180,E1 30841.288,E2 30841.288} C_VEL
LIN {X 0,Y 673.505,Z 786.733,A -85,B 0,C 180,E1 30840.175,E2 30840.175} C_VEL
LIN {X 0,Y 674.376,Z 767.681,A -85,B 0,C 180,E1 30839.432,E2 30839.432} C_VEL
LIN {X 0,Y 675.344,Z 744.914,A -85,B 0,C 180,E1 30838.681,E2 30838.681} C_VEL
LIN {X 0,Y 676.124,Z 721.009,A -85,B 0,C 180,E1 30838.069,E2 30838.069} C_VEL
LIN {X 0,Y 676.788,Z 698.224,A -85,B 0,C 180,E1 30837.624,E2 30837.624} C_VEL
LIN {X 0,Y 677.267,Z 664.299,A -85,B 0,C 180,E1 30837.177,E2 30837.177} C_VEL
LIN {X 0,Y 678.641,Z 503.836,A -85,B 0,C 180,E1 30835.287,E2 30835.287} C_VEL
LIN {X 0,Y 679.056,Z 314.132,A -85,B 0,C 180,E1 30833.179,E2 30833.179} C_VEL
LIN {X 0,Y 677.02,Z 302.362,A -85,B 0,C 180,E1 30832.945,E2 30832.945} C_VEL
LIN {X 0,Y 678.296,Z 263.394,A -85,B 0,C 180,E1 30831.045,E2 30831.045} C_VEL
LIN {X 0,Y 680.073,Z 235.309,A -85,B 0,C 180,E1 30829.541,E2 30829.541} C_VEL
LIN {X 0,Y 674.941,Z 223.486,A -85,B 0,C 180,E1 30828.301,E2 30828.301} C_VEL
LIN {X 0,Y 671.142,Z 215.513,A -85,B 0,C 180,E1 30827.264,E2 30827.264} C_VEL
LIN {X 0,Y 669.286,Z 211.675,A -85,B 0,C 180,E1 30826.683,E2 30826.683} C_VEL
LIN {X 0,Y 667.505,Z 208.267,A -85,B 0,C 180,E1 30826.088,E2 30826.088} C_VEL
LIN {X 0,Y 666.66,Z 206.857,A -85,B 0,C 180,E1 30825.802,E2 30825.802} C_VEL
LIN {X 0,Y 664.748,Z 203.215,A -85,B 0,C 180,E1 30824.988,E2 30824.988} C_VEL
LIN {X 0,Y 664.604,Z 202.447,A -85,B 0,C 180,E1 30824.824,E2 30824.824} C_VEL
LIN {X 0,Y 664.63,Z 202.445,A -85,B 0,C 180,E1 30821.911,E2 30821.911} C_VEL
LIN {X 0,Y 664.619,Z 202.542,A -85,B 0,C 180,E1 30818.856,E2 30818.856} C_VEL
LIN {X 0,Y 666.113,Z 206.162,A -85,B 0,C 180,E1 30818.094,E2 30818.094} C_VEL
LIN {X 0,Y 667.299,Z 207.884,A -85,B 0,C 180,E1 30817.706,E2 30817.706} C_VEL
LIN {X 0,Y 669.667,Z 213.106,A -85,B 0,C 180,E1 30816.84,E2 30816.84} C_VEL
LIN {X 0,Y 672.856,Z 220.2,A -85,B 0,C 180,E1 30815.839,E2 30815.839} C_VEL
LIN {X 0,Y 677.01,Z 231.189,A -85,B 0,C 180,E1 30814.568,E2 30814.568} C_VEL
LIN {X 0,Y 673.983,Z 271.912,A -85,B 0,C 180,E1 30811.88,E2 30811.88} C_VEL
LIN {X 0,Y 671.543,Z 323.07,A -85,B 0,C 180,E1 30808.698,E2 30808.698} C_VEL
LIN {X 0,Y 669.914,Z 373.381,A -85,B 0,C 180,E1 30805.696,E2 30805.696} C_VEL
LIN {X 0,Y 668.512,Z 427.545,A -85,B 0,C 180,E1 30802.56,E2 30802.56} C_VEL
LIN {X 0,Y 668.026,Z 454.865,A -85,B 0,C 180,E1 30801.031,E2 30801.031} C_VEL
LIN {X 0,Y 671.143,Z 482.14,A -85,B 0,C 180,E1 30800.463,E2 30800.463} C_VEL
LIN {X 0,Y 668.827,Z 611.23,A -85,B 0,C 180,E1 30798.748,E2 30798.748} C_VEL
LIN {X 0,Y 668.046,Z 682.529,A -85,B 0,C 180,E1 30797.836,E2 30797.836} C_VEL
LIN {X 0,Y 667.722,Z 702.22,A -85,B 0,C 180,E1 30797.424,E2 30797.424} C_VEL
LIN {X 0,Y 667.369,Z 720.269,A -85,B 0,C 180,E1 30796.898,E2 30796.898} C_VEL
LIN {X 0,Y 666.928,Z 738.747,A -85,B 0,C 180,E1 30796.192,E2 30796.192} C_VEL
LIN {X 0,Y 666.499,Z 756.092,A -85,B 0,C 180,E1 30795.354,E2 30795.354} C_VEL
LIN {X 0,Y 666.055,Z 772.357,A -85,B 0,C 180,E1 30794.386,E2 30794.386} C_VEL
LIN {X 0,Y 665.628,Z 786.962,A -85,B 0,C 180,E1 30793.332,E2 30793.332} C_VEL
LIN {X 0,Y 665.228,Z 800.57,A -85,B 0,C 180,E1 30792.148,E2 30792.148} C_VEL
LIN {X 0,Y 664.886,Z 812.622,A -85,B 0,C 180,E1 30790.882,E2 30790.882} C_VEL
LIN {X 0,Y 664.596,Z 823.273,A -85,B 0,C 180,E1 30789.526,E2 30789.526} C_VEL
LIN {X 0,Y 664.372,Z 832.203,A -85,B 0,C 180,E1 30788.133,E2 30788.133} C_VEL
LIN {X 0,Y 664.22,Z 839.764,A -85,B 0,C 180,E1 30786.656,E2 30786.656} C_VEL
LIN {X 0,Y 664.134,Z 845.878,A -85,B 0,C 180,E1 30785.096,E2 30785.096} C_VEL
LIN {X 0,Y 664.059,Z 850.44,A -85,B 0,C 180,E1 30783.453,E2 30783.453} C_VEL
LIN {X 0,Y 664.028,Z 853.189,A -85,B 0,C 180,E1 30781.812,E2 30781.812} C_VEL
LIN {X 0,Y 664.017,Z 854.212,A -85,B 0,C 180,E1 30780.173,E2 30780.173} C_VEL
LIN {X 0,Y 664.009,Z 853.537,A -85,B 0,C 180,E1 30778.533,E2 30778.533} C_VEL
LIN {X 0,Y 664.027,Z 851.145,A -85,B 0,C 180,E1 30776.893,E2 30776.893} C_VEL
LIN {X 0,Y 664.059,Z 846.969,A -85,B 0,C 180,E1 30775.25,E2 30775.25} C_VEL
LIN {X 0,Y 664.132,Z 841.242,A -85,B 0,C 180,E1 30773.69,E2 30773.69} C_VEL
LIN {X 0,Y 664.255,Z 833.626,A -85,B 0,C 180,E1 30772.127,E2 30772.127} C_VEL
LIN {X 0,Y 664.456,Z 824.453,A -85,B 0,C 180,E1 30770.647,E2 30770.647} C_VEL
LIN {X 0,Y 664.725,Z 813.761,A -85,B 0,C 180,E1 30769.25,E2 30769.25} C_VEL
LIN {X 0,Y 665.06,Z 801.543,A -85,B 0,C 180,E1 30767.937,E2 30767.937} C_VEL
LIN {X 0,Y 665.464,Z 787.735,A -85,B 0,C 180,E1 30766.709,E2 30766.709} C_VEL
LIN {X 0,Y 665.907,Z 772.827,A -85,B 0,C 180,E1 30765.611,E2 30765.611} C_VEL
LIN {X 0,Y 666.365,Z 756.903,A -85,B 0,C 180,E1 30764.642,E2 30764.642} C_VEL
LIN {X 0,Y 666.799,Z 740.025,A -85,B 0,C 180,E1 30763.805,E2 30763.805} C_VEL
LIN {X 0,Y 667.255,Z 722.177,A -85,B 0,C 180,E1 30763.099,E2 30763.099} C_VEL
LIN {X 0,Y 667.644,Z 702.845,A -85,B 0,C 180,E1 30762.518,E2 30762.518} C_VEL
LIN {X 0,Y 667.965,Z 683.249,A -85,B 0,C 180,E1 30762.104,E2 30762.104} C_VEL
LIN {X 0,Y 668.246,Z 651.707,A -85,B 0,C 180,E1 30761.702,E2 30761.702} C_VEL
LIN {X 0,Y 669.337,Z 527.67,A -85,B 0,C 180,E1 30760.25,E2 30760.25} C_VEL
LIN {X 0,Y 668.499,Z 520.085,A -85,B 0,C 180,E1 30760.127,E2 30760.127} C_VEL
LIN {X 0,Y 662.906,Z 500.254,A -85,B 0,C 180,E1 30759.679,E2 30759.679} C_VEL
LIN {X 0,Y 662.276,Z 493.734,A -85,B 0,C 180,E1 30759.574,E2 30759.574} C_VEL
LIN {X 0,Y 662.163,Z 479.253,A -85,B 0,C 180,E1 30759.389,E2 30759.389} C_VEL
LIN {X 0,Y 660.317,Z 463.951,A -85,B 0,C 180,E1 30759.115,E2 30759.115} C_VEL
LIN {X 0,Y 661.651,Z 408.238,A -85,B 0,C 180,E1 30755.919,E2 30755.919} C_VEL
LIN {X 0,Y 663.089,Z 354.866,A -85,B 0,C 180,E1 30752.812,E2 30752.812} C_VEL
LIN {X 0,Y 664.656,Z 302.168,A -85,B 0,C 180,E1 30749.687,E2 30749.687} C_VEL
LIN {X 0,Y 666.284,Z 251.53,A -85,B 0,C 180,E1 30746.632,E2 30746.632} C_VEL
LIN {X 0,Y 666.861,Z 230.371,A -85,B 0,C 180,E1 30745.328,E2 30745.328} C_VEL
LIN {X 0,Y 657.644,Z 206.367,A -85,B 0,C 180,E1 30743.251,E2 30743.251} C_VEL
LIN {X 0,Y 656.679,Z 203.425,A -85,B 0,C 180,E1 30742.972,E2 30742.972} C_VEL
LIN {X 0,Y 656.639,Z 203.437,A -85,B 0,C 180,E1 30739.786,E2 30739.786} C_VEL
LIN {X 0,Y 656.707,Z 203.429,A -85,B 0,C 180,E1 30736.957,E2 30736.957} C_VEL
LIN {X 0,Y 656.698,Z 203.431,A -85,B 0,C 180,E1 30733.851,E2 30733.851} C_VEL
LIN {X 0,Y 656.67,Z 203.429,A -85,B 0,C 180,E1 30730.901,E2 30730.901} C_VEL
LIN {X 0,Y 656.659,Z 203.571,A -85,B 0,C 180,E1 30727.788,E2 30727.788} C_VEL
LIN {X 0,Y 659.411,Z 210.425,A -85,B 0,C 180,E1 30727.171,E2 30727.171} C_VEL
LIN {X 0,Y 666.925,Z 229.465,A -85,B 0,C 180,E1 30725.353,E2 30725.353} C_VEL
LIN {X 0,Y 668.197,Z 233.521,A -85,B 0,C 180,E1 30724.968,E2 30724.968} C_VEL
LIN {X 0,Y 666.824,Z 271.489,A -85,B 0,C 180,E1 30722.162,E2 30722.162} C_VEL
LIN {X 0,Y 665.888,Z 314.948,A -85,B 0,C 180,E1 30719.1,E2 30719.1} C_VEL
LIN {X 0,Y 667.246,Z 323.21,A -85,B 0,C 180,E1 30718.931,E2 30718.931} C_VEL
LIN {X 0,Y 664.264,Z 610.518,A -85,B 0,C 180,E1 30715.492,E2 30715.492} C_VEL
LIN {X 0,Y 663.816,Z 633.766,A -85,B 0,C 180,E1 30715.056,E2 30715.056} C_VEL
LIN {X 0,Y 663.244,Z 654.864,A -85,B 0,C 180,E1 30714.493,E2 30714.493} C_VEL
LIN {X 0,Y 662.667,Z 672.683,A -85,B 0,C 180,E1 30713.895,E2 30713.895} C_VEL
LIN {X 0,Y 661.959,Z 691.537,A -85,B 0,C 180,E1 30713.125,E2 30713.125} C_VEL
LIN {X 0,Y 661.069,Z 712.535,A -85,B 0,C 180,E1 30712.078,E2 30712.078} C_VEL
LIN {X 0,Y 660.244,Z 729.899,A -85,B 0,C 180,E1 30711.034,E2 30711.034} C_VEL
LIN {X 0,Y 659.542,Z 744.37,A -85,B 0,C 180,E1 30710.037,E2 30710.037} C_VEL
LIN {X 0,Y 658.871,Z 758.265,A -85,B 0,C 180,E1 30708.951,E2 30708.951} C_VEL
LIN {X 0,Y 658.262,Z 771.53,A -85,B 0,C 180,E1 30707.777,E2 30707.777} C_VEL
LIN {X 0,Y 657.696,Z 784.093,A -85,B 0,C 180,E1 30706.517,E2 30706.517} C_VEL
LIN {X 0,Y 657.144,Z 798.156,A -85,B 0,C 180,E1 30704.901,E2 30704.901} C_VEL
LIN {X 0,Y 656.69,Z 810.559,A -85,B 0,C 180,E1 30703.203,E2 30703.203} C_VEL
LIN {X 0,Y 656.397,Z 820.029,A -85,B 0,C 180,E1 30701.689,E2 30701.689} C_VEL
LIN {X 0,Y 656.196,Z 828.283,A -85,B 0,C 180,E1 30700.147,E2 30700.147} C_VEL
LIN {X 0,Y 656.053,Z 835.862,A -85,B 0,C 180,E1 30698.449,E2 30698.449} C_VEL
LIN {X 0,Y 655.959,Z 843.283,A -85,B 0,C 180,E1 30696.301,E2 30696.301} C_VEL
LIN {X 0,Y 655.92,Z 847.65,A -85,B 0,C 180,E1 30694.547,E2 30694.547} C_VEL
LIN {X 0,Y 655.905,Z 850.476,A -85,B 0,C 180,E1 30692.884,E2 30692.884} C_VEL
LIN {X 0,Y 655.898,Z 852.06,A -85,B 0,C 180,E1 30691.223,E2 30691.223} C_VEL
LIN {X 0,Y 655.904,Z 852.382,A -85,B 0,C 180,E1 30689.301,E2 30689.301} C_VEL
LIN {X 0,Y 655.911,Z 850.835,A -85,B 0,C 180,E1 30687.291,E2 30687.291} C_VEL
LIN {X 0,Y 655.924,Z 848.191,A -85,B 0,C 180,E1 30685.629,E2 30685.629} C_VEL
LIN {X 0,Y 655.948,Z 844.251,A -85,B 0,C 180,E1 30683.963,E2 30683.963} C_VEL
LIN {X 0,Y 655.99,Z 839.276,A -85,B 0,C 180,E1 30682.38,E2 30682.38} C_VEL
LIN {X 0,Y 656.11,Z 832.323,A -85,B 0,C 180,E1 30680.615,E2 30680.615} C_VEL
LIN {X 0,Y 656.327,Z 822.587,A -85,B 0,C 180,E1 30678.666,E2 30678.666} C_VEL
LIN {X 0,Y 656.604,Z 812.912,A -85,B 0,C 180,E1 30677.065,E2 30677.065} C_VEL
LIN {X 0,Y 656.952,Z 802.902,A -85,B 0,C 180,E1 30675.636,E2 30675.636} C_VEL
LIN {X 0,Y 657.396,Z 791.362,A -85,B 0,C 180,E1 30674.201,E2 30674.201} C_VEL
LIN {X 0,Y 658.061,Z 776.312,A -85,B 0,C 180,E1 30672.583,E2 30672.583} C_VEL
LIN {X 0,Y 658.776,Z 760.413,A -85,B 0,C 180,E1 30671.138,E2 30671.138} C_VEL
LIN {X 0,Y 659.421,Z 746.783,A -85,B 0,C 180,E1 30670.052,E2 30670.052} C_VEL
LIN {X 0,Y 660.109,Z 732.618,A -85,B 0,C 180,E1 30669.055,E2 30669.055} C_VEL
LIN {X 0,Y 660.808,Z 717.967,A -85,B 0,C 180,E1 30668.147,E2 30668.147} C_VEL
LIN {X 0,Y 661.452,Z 703.66,A -85,B 0,C 180,E1 30667.369,E2 30667.369} C_VEL
LIN {X 0,Y 662.067,Z 688.3,A -85,B 0,C 180,E1 30666.644,E2 30666.644} C_VEL
LIN {X 0,Y 662.768,Z 669.972,A -85,B 0,C 180,E1 30665.915,E2 30665.915} C_VEL
LIN {X 0,Y 663.459,Z 648.459,A -85,B 0,C 180,E1 30665.224,E2 30665.224} C_VEL
LIN {X 0,Y 663.992,Z 625.89,A -85,B 0,C 180,E1 30664.686,E2 30664.686} C_VEL
LIN {X 0,Y 664.319,Z 605.36,A -85,B 0,C 180,E1 30664.347,E2 30664.347} C_VEL
LIN {X 0,Y 667.251,Z 321.851,A -85,B 0,C 180,E1 30660.961,E2 30660.961} C_VEL
LIN {X 0,Y 665.89,Z 314.577,A -85,B 0,C 180,E1 30660.79,E2 30660.79} C_VEL
LIN {X 0,Y 666.879,Z 269.958,A -85,B 0,C 180,E1 30657.638,E2 30657.638} C_VEL
LIN {X 0,Y 668.183,Z 233.072,A -85,B 0,C 180,E1 30654.907,E2 30654.907} C_VEL
LIN {X 0,Y 661.541,Z 215.766,A -85,B 0,C 180,E1 30653.233,E2 30653.233} C_VEL
LIN {X 0,Y 656.721,Z 203.547,A -85,B 0,C 180,E1 30652.121,E2 30652.121} C_VEL
LIN {X 0,Y 656.677,Z 203.427,A -85,B 0,C 180,E1 30649.046,E2 30649.046} C_VEL
LIN {X 0,Y 656.703,Z 203.428,A -85,B 0,C 180,E1 30646.028,E2 30646.028} C_VEL
LIN {X 0,Y 656.68,Z 203.425,A -85,B 0,C 180,E1 30643.012,E2 30643.012} C_VEL
LIN {X 0,Y 656.699,Z 203.427,A -85,B 0,C 180,E1 30640.016,E2 30640.016} C_VEL
LIN {X 0,Y 656.683,Z 203.424,A -85,B 0,C 180,E1 30636.929,E2 30636.929} C_VEL
LIN {X 0,Y 656.696,Z 203.423,A -85,B 0,C 180,E1 30633.92,E2 30633.92} C_VEL
LIN {X 0,Y 656.687,Z 203.427,A -85,B 0,C 180,E1 30630.872,E2 30630.872} C_VEL
LIN {X 0,Y 656.694,Z 203.424,A -85,B 0,C 180,E1 30627.869,E2 30627.869} C_VEL
LIN {X 0,Y 656.69,Z 203.425,A -85,B 0,C 180,E1 30624.84,E2 30624.84} C_VEL
LIN {X 0,Y 656.692,Z 203.427,A -85,B 0,C 180,E1 30621.809,E2 30621.809} C_VEL
LIN {X 0,Y 656.693,Z 203.421,A -85,B 0,C 180,E1 30618.74,E2 30618.74} C_VEL
LIN {X 0,Y 656.687,Z 203.427,A -85,B 0,C 180,E1 30615.726,E2 30615.726} C_VEL
LIN {X 0,Y 656.695,Z 203.418,A -85,B 0,C 180,E1 30612.755,E2 30612.755} C_VEL
LIN {X 0,Y 656.685,Z 203.428,A -85,B 0,C 180,E1 30609.73,E2 30609.73} C_VEL
LIN {X 0,Y 656.697,Z 203.419,A -85,B 0,C 180,E1 30606.733,E2 30606.733} C_VEL
LIN {X 0,Y 656.682,Z 203.428,A -85,B 0,C 180,E1 30603.667,E2 30603.667} C_VEL
LIN {X 0,Y 656.698,Z 203.424,A -85,B 0,C 180,E1 30600.611,E2 30600.611} C_VEL
LIN {X 0,Y 656.677,Z 203.427,A -85,B 0,C 180,E1 30597.644,E2 30597.644} C_VEL
LIN {X 0,Y 656.701,Z 203.426,A -85,B 0,C 180,E1 30594.583,E2 30594.583} C_VEL
LIN {X 0,Y 656.674,Z 203.424,A -85,B 0,C 180,E1 30591.595,E2 30591.595} C_VEL
LIN {X 0,Y 656.703,Z 203.426,A -85,B 0,C 180,E1 30588.584,E2 30588.584} C_VEL
LIN {X 0,Y 656.671,Z 203.427,A -85,B 0,C 180,E1 30585.539,E2 30585.539} C_VEL
LIN {X 0,Y 656.706,Z 203.427,A -85,B 0,C 180,E1 30582.545,E2 30582.545} C_VEL
LIN {X 0,Y 656.669,Z 203.428,A -85,B 0,C 180,E1 30579.499,E2 30579.499} C_VEL
LIN {X 0,Y 656.708,Z 203.428,A -85,B 0,C 180,E1 30576.489,E2 30576.489} C_VEL
LIN {X 0,Y 656.665,Z 203.427,A -85,B 0,C 180,E1 30573.503,E2 30573.503} C_VEL
LIN {X 0,Y 656.711,Z 203.425,A -85,B 0,C 180,E1 30570.541,E2 30570.541} C_VEL
LIN {X 0,Y 656.661,Z 203.432,A -85,B 0,C 180,E1 30567.486,E2 30567.486} C_VEL
LIN {X 0,Y 656.708,Z 203.427,A -85,B 0,C 180,E1 30564.542,E2 30564.542} C_VEL
LIN {X 0,Y 656.658,Z 203.433,A -85,B 0,C 180,E1 30561.48,E2 30561.48} C_VEL
LIN {X 0,Y 656.713,Z 203.427,A -85,B 0,C 180,E1 30558.513,E2 30558.513} C_VEL
LIN {X 0,Y 656.655,Z 203.434,A -85,B 0,C 180,E1 30555.449,E2 30555.449} C_VEL
LIN {X 0,Y 656.733,Z 203.614,A -85,B 0,C 180,E1 30554.09,E2 30554.09} C_VEL
LIN {X 0,Y 657.964,Z 206.886,A -85,B 0,C 180,E1 30553.793,E2 30553.793} C_VEL
LIN {X 0,Y 666.705,Z 224.357,A -85,B 0,C 180,E1 30552.065,E2 30552.065} C_VEL
LIN {X 0,Y 673.617,Z 239.079,A -85,B 0,C 180,E1 30550.743,E2 30550.743} C_VEL
LIN {X 0,Y 671.5,Z 291.807,A -85,B 0,C 180,E1 30548.112,E2 30548.112} C_VEL
LIN {X 0,Y 671.164,Z 302.005,A -85,B 0,C 180,E1 30547.625,E2 30547.625} C_VEL
LIN {X 0,Y 673.391,Z 317.785,A -85,B 0,C 180,E1 30547.284,E2 30547.284} C_VEL
LIN {X 0,Y 671.173,Z 579.716,A -85,B 0,C 180,E1 30544.173,E2 30544.173} C_VEL
LIN {X 0,Y 670.199,Z 688.285,A -85,B 0,C 180,E1 30542.892,E2 30542.892} C_VEL
LIN {X 0,Y 669.641,Z 712.806,A -85,B 0,C 180,E1 30542.476,E2 30542.476} C_VEL
LIN {X 0,Y 668.783,Z 735.948,A -85,B 0,C 180,E1 30541.924,E2 30541.924} C_VEL
LIN {X 0,Y 667.921,Z 756.984,A -85,B 0,C 180,E1 30541.296,E2 30541.296} C_VEL
LIN {X 0,Y 666.738,Z 780.733,A -85,B 0,C 180,E1 30540.422,E2 30540.422} C_VEL
LIN {X 0,Y 665.734,Z 800.161,A -85,B 0,C 180,E1 30539.568,E2 30539.568} C_VEL
LIN {X 0,Y 664.477,Z 822.251,A -85,B 0,C 180,E1 30538.442,E2 30538.442} C_VEL
LIN {X 0,Y 663.221,Z 842.297,A -85,B 0,C 180,E1 30537.245,E2 30537.245} C_VEL
LIN {X 0,Y 662.03,Z 862.353,A -85,B 0,C 180,E1 30535.88,E2 30535.88} C_VEL
LIN {X 0,Y 660.824,Z 881.181,A -85,B 0,C 180,E1 30534.398,E2 30534.398} C_VEL
LIN {X 0,Y 659.791,Z 898.888,A -85,B 0,C 180,E1 30532.828,E2 30532.828} C_VEL
LIN {X 0,Y 658.834,Z 915.095,A -85,B 0,C 180,E1 30531.174,E2 30531.174} C_VEL
LIN {X 0,Y 658.029,Z 930.99,A -85,B 0,C 180,E1 30529.345,E2 30529.345} C_VEL
LIN {X 0,Y 657.344,Z 944.842,A -85,B 0,C 180,E1 30527.496,E2 30527.496} C_VEL
LIN {X 0,Y 656.828,Z 957.687,A -85,B 0,C 180,E1 30525.541,E2 30525.541} C_VEL
LIN {X 0,Y 656.443,Z 968.646,A -85,B 0,C 180,E1 30523.566,E2 30523.566} C_VEL
LIN {X 0,Y 656.206,Z 977.993,A -85,B 0,C 180,E1 30521.603,E2 30521.603} C_VEL
LIN {X 0,Y 656.049,Z 985.907,A -85,B 0,C 180,E1 30519.563,E2 30519.563} C_VEL
LIN {X 0,Y 655.943,Z 991.744,A -85,B 0,C 180,E1 30517.709,E2 30517.709} C_VEL
LIN {X 0,Y 655.912,Z 996.857,A -85,B 0,C 180,E1 30515.599,E2 30515.599} C_VEL
LIN {X 0,Y 655.914,Z 1000.012,A -85,B 0,C 180,E1 30513.671,E2 30513.671} C_VEL
LIN {X 0,Y 655.9,Z 1001.968,A -85,B 0,C 180,E1 30511.66,E2 30511.66} C_VEL
LIN {X 0,Y 655.885,Z 1002.395,A -85,B 0,C 180,E1 30509.563,E2 30509.563} C_VEL
LIN {X 0,Y 655.914,Z 1001.498,A -85,B 0,C 180,E1 30507.728,E2 30507.728} C_VEL
LIN {X 0,Y 655.92,Z 998.919,A -85,B 0,C 180,E1 30505.538,E2 30505.538} C_VEL
LIN {X 0,Y 655.93,Z 994.895,A -85,B 0,C 180,E1 30503.523,E2 30503.523} C_VEL
LIN {X 0,Y 655.985,Z 989.71,A -85,B 0,C 180,E1 30501.586,E2 30501.586} C_VEL
LIN {X 0,Y 656.122,Z 982.073,A -85,B 0,C 180,E1 30499.403,E2 30499.403} C_VEL
LIN {X 0,Y 656.307,Z 974.248,A -85,B 0,C 180,E1 30497.574,E2 30497.574} C_VEL
LIN {X 0,Y 656.637,Z 963.38,A -85,B 0,C 180,E1 30495.448,E2 30495.448} C_VEL
LIN {X 0,Y 657.027,Z 952.549,A -85,B 0,C 180,E1 30493.648,E2 30493.648} C_VEL
LIN {X 0,Y 657.641,Z 938.726,A -85,B 0,C 180,E1 30491.656,E2 30491.656} C_VEL
LIN {X 0,Y 658.309,Z 924.852,A -85,B 0,C 180,E1 30489.924,E2 30489.924} C_VEL
LIN {X 0,Y 659.245,Z 908.158,A -85,B 0,C 180,E1 30488.092,E2 30488.092} C_VEL
LIN {X 0,Y 660.181,Z 891.811,A -85,B 0,C 180,E1 30486.526,E2 30486.526} C_VEL
LIN {X 0,Y 661.369,Z 872.641,A -85,B 0,C 180,E1 30484.905,E2 30484.905} C_VEL
LIN {X 0,Y 662.48,Z 854.399,A -85,B 0,C 180,E1 30483.561,E2 30483.561} C_VEL
LIN {X 0,Y 663.804,Z 833.587,A -85,B 0,C 180,E1 30482.212,E2 30482.212} C_VEL
LIN {X 0,Y 664.99,Z 812.835,A -85,B 0,C 180,E1 30481.058,E2 30481.058} C_VEL
LIN {X 0,Y 666.28,Z 790.543,A -85,B 0,C 180,E1 30479.987,E2 30479.987} C_VEL
LIN {X 0,Y 667.346,Z 768.964,A -85,B 0,C 180,E1 30479.125,E2 30479.125} C_VEL
LIN {X 0,Y 668.306,Z 748.103,A -85,B 0,C 180,E1 30478.422,E2 30478.422} C_VEL
LIN {X 0,Y 669.246,Z 722.705,A -85,B 0,C 180,E1 30477.743,E2 30477.743} C_VEL
LIN {X 0,Y 669.927,Z 700.955,A -85,B 0,C 180,E1 30477.305,E2 30477.305} C_VEL
LIN {X 0,Y 670.481,Z 670.013,A -85,B 0,C 180,E1 30476.875,E2 30476.875} C_VEL
LIN {X 0,Y 671.199,Z 531.958,A -85,B 0,C 180,E1 30475.329,E2 30475.329} C_VEL
LIN {X 0,Y 671.916,Z 315.674,A -85,B 0,C 180,E1 30472.901,E2 30472.901} C_VEL
LIN {X 0,Y 669.934,Z 303.804,A -85,B 0,C 180,E1 30472.653,E2 30472.653} C_VEL
LIN {X 0,Y 671.509,Z 265.684,A -85,B 0,C 180,E1 30470.74,E2 30470.74} C_VEL
LIN {X 0,Y 673.601,Z 239.115,A -85,B 0,C 180,E1 30469.27,E2 30469.27} C_VEL
LIN {X 0,Y 668.998,Z 228.301,A -85,B 0,C 180,E1 30468.08,E2 30468.08} C_VEL
LIN {X 0,Y 665.749,Z 221.208,A -85,B 0,C 180,E1 30467.128,E2 30467.128} C_VEL
LIN {X 0,Y 663.628,Z 217.001,A -85,B 0,C 180,E1 30466.446,E2 30466.446} C_VEL
LIN {X 0,Y 661.75,Z 213.116,A -85,B 0,C 180,E1 30465.727,E2 30465.727} C_VEL
LIN {X 0,Y 659.752,Z 209.169,A -85,B 0,C 180,E1 30464.824,E2 30464.824} C_VEL
LIN {X 0,Y 657.358,Z 205.737,A -85,B 0,C 180,E1 30463.485,E2 30463.485} C_VEL
LIN {X 0,Y 656.751,Z 203.76,A -85,B 0,C 180,E1 30462.275,E2 30462.275} C_VEL
LIN {X 0,Y 656.789,Z 203.918,A -85,B 0,C 180,E1 30461.231,E2 30461.231} C_VEL
LIN {X 0,Y 657.572,Z 206.261,A -85,B 0,C 180,E1 30459.971,E2 30459.971} C_VEL
LIN {X 0,Y 659.559,Z 208.782,A -85,B 0,C 180,E1 30458.949,E2 30458.949} C_VEL
LIN {X 0,Y 661.234,Z 212.555,A -85,B 0,C 180,E1 30458.095,E2 30458.095} C_VEL
LIN {X 0,Y 662.091,Z 214.188,A -85,B 0,C 180,E1 30457.759,E2 30457.759} C_VEL
LIN {X 0,Y 663.998,Z 218.269,A -85,B 0,C 180,E1 30457.038,E2 30457.038} C_VEL
LIN {X 0,Y 667.432,Z 226.435,A -85,B 0,C 180,E1 30455.857,E2 30455.857} C_VEL
LIN {X 0,Y 670.543,Z 235.099,A -85,B 0,C 180,E1 30454.828,E2 30454.828} C_VEL
LIN {X 0,Y 667.26,Z 273.364,A -85,B 0,C 180,E1 30452.24,E2 30452.24} C_VEL
LIN {X 0,Y 664.493,Z 323.109,A -85,B 0,C 180,E1 30449.08,E2 30449.08} C_VEL
LIN {X 0,Y 662.644,Z 372.235,A -85,B 0,C 180,E1 30446.095,E2 30446.095} C_VEL
LIN {X 0,Y 661.052,Z 426.481,A -85,B 0,C 180,E1 30442.904,E2 30442.904} C_VEL
LIN {X 0,Y 660.499,Z 452.198,A -85,B 0,C 180,E1 30441.438,E2 30441.438} C_VEL
LIN {X 0,Y 664.049,Z 483.157,A -85,B 0,C 180,E1 30440.772,E2 30440.772} C_VEL
LIN {X 0,Y 661.565,Z 600.11,A -85,B 0,C 180,E1 30439.151,E2 30439.151} C_VEL
LIN {X 0,Y 660.467,Z 682.887,A -85,B 0,C 180,E1 30438.055,E2 30438.055} C_VEL
LIN {X 0,Y 660.109,Z 702.739,A -85,B 0,C 180,E1 30437.632,E2 30437.632} C_VEL
LIN {X 0,Y 659.696,Z 722.032,A -85,B 0,C 180,E1 30437.055,E2 30437.055} C_VEL
LIN {X 0,Y 659.228,Z 740.269,A -85,B 0,C 180,E1 30436.341,E2 30436.341} C_VEL
LIN {X 0,Y 658.773,Z 757.486,A -85,B 0,C 180,E1 30435.494,E2 30435.494} C_VEL
LIN {X 0,Y 658.3,Z 773.688,A -85,B 0,C 180,E1 30434.514,E2 30434.514} C_VEL
LIN {X 0,Y 657.845,Z 788.259,A -85,B 0,C 180,E1 30433.447,E2 30433.447} C_VEL
LIN {X 0,Y 657.43,Z 801.382,A -85,B 0,C 180,E1 30432.294,E2 30432.294} C_VEL
LIN {X 0,Y 657.065,Z 813.378,A -85,B 0,C 180,E1 30431.028,E2 30431.028} C_VEL
LIN {X 0,Y 656.748,Z 824.232,A -85,B 0,C 180,E1 30429.641,E2 30429.641} C_VEL
LIN {X 0,Y 656.503,Z 833.218,A -85,B 0,C 180,E1 30428.231,E2 30428.231} C_VEL
LIN {X 0,Y 656.333,Z 840.813,A -85,B 0,C 180,E1 30426.737,E2 30426.737} C_VEL
LIN {X 0,Y 656.229,Z 846.946,A -85,B 0,C 180,E1 30425.158,E2 30425.158} C_VEL
LIN {X 0,Y 656.142,Z 851.513,A -85,B 0,C 180,E1 30423.495,E2 30423.495} C_VEL
LIN {X 0,Y 656.102,Z 854.253,A -85,B 0,C 180,E1 30421.834,E2 30421.834} C_VEL
LIN {X 0,Y 656.085,Z 855.253,A -85,B 0,C 180,E1 30420.175,E2 30420.175} C_VEL
LIN {X 0,Y 656.073,Z 854.541,A -85,B 0,C 180,E1 30418.515,E2 30418.515} C_VEL
LIN {X 0,Y 656.091,Z 852.104,A -85,B 0,C 180,E1 30416.855,E2 30416.855} C_VEL
LIN {X 0,Y 656.129,Z 847.874,A -85,B 0,C 180,E1 30415.192,E2 30415.192} C_VEL
LIN {X 0,Y 656.21,Z 842.087,A -85,B 0,C 180,E1 30413.614,E2 30413.614} C_VEL
LIN {X 0,Y 656.349,Z 834.406,A -85,B 0,C 180,E1 30412.031,E2 30412.031} C_VEL
LIN {X 0,Y 656.569,Z 825.163,A -85,B 0,C 180,E1 30410.533,E2 30410.533} C_VEL
LIN {X 0,Y 656.862,Z 814.399,A -85,B 0,C 180,E1 30409.12,E2 30409.12} C_VEL
LIN {X 0,Y 657.227,Z 802.111,A -85,B 0,C 180,E1 30407.791,E2 30407.791} C_VEL
LIN {X 0,Y 657.662,Z 788.222,A -85,B 0,C 180,E1 30406.549,E2 30406.549} C_VEL
LIN {X 0,Y 658.121,Z 773.911,A -85,B 0,C 180,E1 30405.482,E2 30405.482} C_VEL
LIN {X 0,Y 658.613,Z 758.073,A -85,B 0,C 180,E1 30404.502,E2 30404.502} C_VEL
LIN {X 0,Y 659.072,Z 741.635,A -85,B 0,C 180,E1 30403.668,E2 30403.668} C_VEL
LIN {X 0,Y 659.568,Z 723.742,A -85,B 0,C 180,E1 30402.942,E2 30402.942} C_VEL
LIN {X 0,Y 659.981,Z 704.927,A -85,B 0,C 180,E1 30402.356,E2 30402.356} C_VEL
LIN {X 0,Y 660.339,Z 685.589,A -85,B 0,C 180,E1 30401.925,E2 30401.925} C_VEL
LIN {X 0,Y 660.619,Z 659.994,A -85,B 0,C 180,E1 30401.574,E2 30401.574} C_VEL
LIN {X 0,Y 662.276,Z 493.734,A -85,B 0,C 180,E1 30399.574,E2 30399.574} C_VEL
LIN {X 0,Y 661.35,Z 488.762,A -85,B 0,C 180,E1 30399.477,E2 30399.477} C_VEL
LIN {X 0,Y 654.524,Z 475.181,A -85,B 0,C 180,E1 30399.045,E2 30399.045} C_VEL
LIN {X 0,Y 653.858,Z 472.31,A -85,B 0,C 180,E1 30398.983,E2 30398.983} C_VEL
LIN {X 0,Y 652.75,Z 463.022,A -85,B 0,C 180,E1 30398.807,E2 30398.807} C_VEL
LIN {X 0,Y 654.174,Z 408.167,A -85,B 0,C 180,E1 30395.626,E2 30395.626} C_VEL
LIN {X 0,Y 655.734,Z 355.483,A -85,B 0,C 180,E1 30392.526,E2 30392.526} C_VEL
LIN {X 0,Y 657.428,Z 302.739,A -85,B 0,C 180,E1 30389.369,E2 30389.369} C_VEL
LIN {X 0,Y 659.179,Z 252.858,A -85,B 0,C 180,E1 30386.329,E2 30386.329} C_VEL
LIN {X 0,Y 659.907,Z 233.936,A -85,B 0,C 180,E1 30385.164,E2 30385.164} C_VEL
LIN {X 0,Y 650.721,Z 210.034,A -85,B 0,C 180,E1 30383.072,E2 30383.072} C_VEL
LIN {X 0,Y 648.77,Z 204.417,A -85,B 0,C 180,E1 30382.569,E2 30382.569} C_VEL
LIN {X 0,Y 648.696,Z 204.426,A -85,B 0,C 180,E1 30379.539,E2 30379.539} C_VEL
LIN {X 0,Y 648.771,Z 204.418,A -85,B 0,C 180,E1 30376.545,E2 30376.545} C_VEL
LIN {X 0,Y 648.761,Z 204.418,A -85,B 0,C 180,E1 30373.424,E2 30373.424} C_VEL
LIN {X 0,Y 648.778,Z 204.419,A -85,B 0,C 180,E1 30370.28,E2 30370.28} C_VEL
LIN {X 0,Y 648.766,Z 204.601,A -85,B 0,C 180,E1 30368.245,E2 30368.245} C_VEL
LIN {X 0,Y 651.485,Z 211.429,A -85,B 0,C 180,E1 30367.631,E2 30367.631} C_VEL
LIN {X 0,Y 659.281,Z 230.843,A -85,B 0,C 180,E1 30365.766,E2 30365.766} C_VEL
LIN {X 0,Y 661.28,Z 236.953,A -85,B 0,C 180,E1 30365.176,E2 30365.176} C_VEL
LIN {X 0,Y 659.905,Z 273.928,A -85,B 0,C 180,E1 30362.438,E2 30362.438} C_VEL
LIN {X 0,Y 659.196,Z 306.565,A -85,B 0,C 180,E1 30360.137,E2 30360.137} C_VEL
LIN {X 0,Y 659.229,Z 317.775,A -85,B 0,C 180,E1 30359.399,E2 30359.399} C_VEL
LIN {X 0,Y 660.287,Z 324.684,A -85,B 0,C 180,E1 30359.259,E2 30359.259} C_VEL
LIN {X 0,Y 657.859,Z 518.202,A -85,B 0,C 180,E1 30356.886,E2 30356.886} C_VEL
LIN {X 0,Y 656.758,Z 614.046,A -85,B 0,C 180,E1 30355.694,E2 30355.694} C_VEL
LIN {X 0,Y 656.299,Z 636.159,A -85,B 0,C 180,E1 30355.255,E2 30355.255} C_VEL
LIN {X 0,Y 655.685,Z 657.491,A -85,B 0,C 180,E1 30354.67,E2 30354.67} C_VEL
LIN {X 0,Y 655.003,Z 677.878,A -85,B 0,C 180,E1 30353.958,E2 30353.958} C_VEL
LIN {X 0,Y 654.138,Z 698.947,A -85,B 0,C 180,E1 30353.036,E2 30353.036} C_VEL
LIN {X 0,Y 653.28,Z 717.337,A -85,B 0,C 180,E1 30352.057,E2 30352.057} C_VEL
LIN {X 0,Y 652.47,Z 733.536,A -85,B 0,C 180,E1 30351.048,E2 30351.048} C_VEL
LIN {X 0,Y 651.674,Z 748.645,A -85,B 0,C 180,E1 30349.962,E2 30349.962} C_VEL
LIN {X 0,Y 650.748,Z 766.708,A -85,B 0,C 180,E1 30348.453,E2 30348.453} C_VEL
LIN {X 0,Y 650.053,Z 780.67,A -85,B 0,C 180,E1 30347.085,E2 30347.085} C_VEL
LIN {X 0,Y 649.515,Z 792.121,A -85,B 0,C 180,E1 30345.812,E2 30345.812} C_VEL
LIN {X 0,Y 649.06,Z 802.897,A -85,B 0,C 180,E1 30344.452,E2 30344.452} C_VEL
LIN {X 0,Y 648.693,Z 812.605,A -85,B 0,C 180,E1 30343.052,E2 30343.052} C_VEL
LIN {X 0,Y 648.408,Z 821.558,A -85,B 0,C 180,E1 30341.564,E2 30341.564} C_VEL
LIN {X 0,Y 648.172,Z 830.734,A -85,B 0,C 180,E1 30339.77,E2 30339.77} C_VEL
LIN {X 0,Y 648.011,Z 838.66,A -85,B 0,C 180,E1 30337.804,E2 30337.804} C_VEL
LIN {X 0,Y 647.956,Z 844,A -85,B 0,C 180,E1 30336.112,E2 30336.112} C_VEL
LIN {X 0,Y 647.925,Z 848.002,A -85,B 0,C 180,E1 30334.425,E2 30334.425} C_VEL
LIN {X 0,Y 647.91,Z 850.709,A -85,B 0,C 180,E1 30332.742,E2 30332.742} C_VEL
LIN {X 0,Y 647.912,Z 852.339,A -85,B 0,C 180,E1 30330.796,E2 30330.796} C_VEL
LIN {X 0,Y 647.901,Z 852.116,A -85,B 0,C 180,E1 30328.762,E2 30328.762} C_VEL
LIN {X 0,Y 647.905,Z 850.593,A -85,B 0,C 180,E1 30327.081,E2 30327.081} C_VEL
LIN {X 0,Y 647.924,Z 848.005,A -85,B 0,C 180,E1 30325.486,E2 30325.486} C_VEL
LIN {X 0,Y 647.958,Z 844.004,A -85,B 0,C 180,E1 30323.799,E2 30323.799} C_VEL
LIN {X 0,Y 648.01,Z 838.663,A -85,B 0,C 180,E1 30322.107,E2 30322.107} C_VEL
LIN {X 0,Y 648.173,Z 830.735,A -85,B 0,C 180,E1 30320.141,E2 30320.141} C_VEL
LIN {X 0,Y 648.408,Z 821.558,A -85,B 0,C 180,E1 30318.345,E2 30318.345} C_VEL
LIN {X 0,Y 648.679,Z 812.902,A -85,B 0,C 180,E1 30316.904,E2 30316.904} C_VEL
LIN {X 0,Y 649.035,Z 803.559,A -85,B 0,C 180,E1 30315.548,E2 30315.548} C_VEL
LIN {X 0,Y 649.481,Z 792.866,A -85,B 0,C 180,E1 30314.187,E2 30314.187} C_VEL
LIN {X 0,Y 650.008,Z 781.506,A -85,B 0,C 180,E1 30312.914,E2 30312.914} C_VEL
LIN {X 0,Y 650.637,Z 768.608,A -85,B 0,C 180,E1 30311.637,E2 30311.637} C_VEL
LIN {X 0,Y 651.548,Z 751.654,A -85,B 0,C 180,E1 30310.175,E2 30310.175} C_VEL
LIN {X 0,Y 652.411,Z 734.668,A -85,B 0,C 180,E1 30308.937,E2 30308.937} C_VEL
LIN {X 0,Y 653.221,Z 718.608,A -85,B 0,C 180,E1 30307.927,E2 30307.927} C_VEL
LIN {X 0,Y 653.96,Z 702.441,A -85,B 0,C 180,E1 30307.052,E2 30307.052} C_VEL
LIN {X 0,Y 654.802,Z 683.002,A -85,B 0,C 180,E1 30306.161,E2 30306.161} C_VEL
LIN {X 0,Y 655.55,Z 661.856,A -85,B 0,C 180,E1 30305.377,E2 30305.377} C_VEL
LIN {X 0,Y 656.187,Z 640.976,A -85,B 0,C 180,E1 30304.771,E2 30304.771} C_VEL
LIN {X 0,Y 656.632,Z 619.434,A -85,B 0,C 180,E1 30304.313,E2 30304.313} C_VEL
LIN {X 0,Y 657.002,Z 593.281,A -85,B 0,C 180,E1 30303.942,E2 30303.942} C_VEL
LIN {X 0,Y 660.174,Z 335.018,A -85,B 0,C 180,E1 30300.773,E2 30300.773} C_VEL
LIN {X 0,Y 660.114,Z 322.291,A -85,B 0,C 180,E1 30300.611,E2 30300.611} C_VEL
LIN {X 0,Y 659.163,Z 317.144,A -85,B 0,C 180,E1 30300.487,E2 30300.487} C_VEL
LIN {X 0,Y 659.693,Z 280.043,A -85,B 0,C 180,E1 30297.917,E2 30297.917} C_VEL
LIN {X 0,Y 661.162,Z 241.324,A -85,B 0,C 180,E1 30295.053,E2 30295.053} C_VEL
LIN {X 0,Y 661.205,Z 236.237,A -85,B 0,C 180,E1 30294.672,E2 30294.672} C_VEL
LIN {X 0,Y 654.289,Z 218.189,A -85,B 0,C 180,E1 30292.914,E2 30292.914} C_VEL
LIN {X 0,Y 648.793,Z 204.584,A -85,B 0,C 180,E1 30291.656,E2 30291.656} C_VEL
LIN {X 0,Y 648.748,Z 204.415,A -85,B 0,C 180,E1 30288.608,E2 30288.608} C_VEL
LIN {X 0,Y 648.762,Z 204.418,A -85,B 0,C 180,E1 30285.402,E2 30285.402} C_VEL
LIN {X 0,Y 648.769,Z 204.424,A -85,B 0,C 180,E1 30282.219,E2 30282.219} C_VEL
LIN {X 0,Y 648.748,Z 204.416,A -85,B 0,C 180,E1 30279.078,E2 30279.078} C_VEL
LIN {X 0,Y 648.761,Z 204.417,A -85,B 0,C 180,E1 30275.987,E2 30275.987} C_VEL
LIN {X 0,Y 648.748,Z 204.408,A -85,B 0,C 180,E1 30272.961,E2 30272.961} C_VEL
LIN {X 0,Y 648.757,Z 204.414,A -85,B 0,C 180,E1 30269.958,E2 30269.958} C_VEL
LIN {X 0,Y 648.753,Z 204.411,A -85,B 0,C 180,E1 30266.945,E2 30266.945} C_VEL
LIN {X 0,Y 648.755,Z 204.403,A -85,B 0,C 180,E1 30263.913,E2 30263.913} C_VEL
LIN {X 0,Y 648.754,Z 204.414,A -85,B 0,C 180,E1 30260.857,E2 30260.857} C_VEL
LIN {X 0,Y 648.752,Z 204.405,A -85,B 0,C 180,E1 30257.861,E2 30257.861} C_VEL
LIN {X 0,Y 648.757,Z 204.413,A -85,B 0,C 180,E1 30254.824,E2 30254.824} C_VEL
LIN {X 0,Y 648.746,Z 204.408,A -85,B 0,C 180,E1 30251.739,E2 30251.739} C_VEL
LIN {X 0,Y 648.758,Z 204.416,A -85,B 0,C 180,E1 30248.687,E2 30248.687} C_VEL
LIN {X 0,Y 648.742,Z 204.405,A -85,B 0,C 180,E1 30245.661,E2 30245.661} C_VEL
LIN {X 0,Y 648.76,Z 204.417,A -85,B 0,C 180,E1 30242.562,E2 30242.562} C_VEL
LIN {X 0,Y 648.738,Z 204.399,A -85,B 0,C 180,E1 30239.558,E2 30239.558} C_VEL
LIN {X 0,Y 648.763,Z 204.416,A -85,B 0,C 180,E1 30236.466,E2 30236.466} C_VEL
LIN {X 0,Y 648.736,Z 204.4,A -85,B 0,C 180,E1 30233.451,E2 30233.451} C_VEL
LIN {X 0,Y 648.765,Z 204.414,A -85,B 0,C 180,E1 30230.418,E2 30230.418} C_VEL
LIN {X 0,Y 648.735,Z 204.415,A -85,B 0,C 180,E1 30227.358,E2 30227.358} C_VEL
LIN {X 0,Y 648.77,Z 204.416,A -85,B 0,C 180,E1 30224.261,E2 30224.261} C_VEL
LIN {X 0,Y 648.735,Z 204.413,A -85,B 0,C 180,E1 30221.208,E2 30221.208} C_VEL
LIN {X 0,Y 648.769,Z 204.417,A -85,B 0,C 180,E1 30218.096,E2 30218.096} C_VEL
LIN {X 0,Y 648.742,Z 204.415,A -85,B 0,C 180,E1 30215.019,E2 30215.019} C_VEL
LIN {X 0,Y 648.738,Z 204.42,A -85,B 0,C 180,E1 30211.759,E2 30211.759} C_VEL
LIN {X 0,Y 648.754,Z 204.415,A -85,B 0,C 180,E1 30208.803,E2 30208.803} C_VEL
LIN {X 0,Y 648.73,Z 204.422,A -85,B 0,C 180,E1 30205.659,E2 30205.659} C_VEL
LIN {X 0,Y 648.759,Z 204.416,A -85,B 0,C 180,E1 30202.681,E2 30202.681} C_VEL
LIN {X 0,Y 648.722,Z 204.424,A -85,B 0,C 180,E1 30199.541,E2 30199.541} C_VEL
LIN {X 0,Y 648.764,Z 204.415,A -85,B 0,C 180,E1 30196.545,E2 30196.545} C_VEL
LIN {X 0,Y 648.754,Z 204.491,A -85,B 0,C 180,E1 30194.709,E2 30194.709} C_VEL
LIN {X 0,Y 649.81,Z 207.478,A -85,B 0,C 180,E1 30194.437,E2 30194.437} C_VEL
LIN {X 0,Y 651.127,Z 209.868,A -85,B 0,C 180,E1 30194.181,E2 30194.181} C_VEL
LIN {X 0,Y 660.682,Z 229.107,A -85,B 0,C 180,E1 30192.263,E2 30192.263} C_VEL
LIN {X 0,Y 667.072,Z 242.765,A -85,B 0,C 180,E1 30191.018,E2 30191.018} C_VEL
LIN {X 0,Y 664.694,Z 294.604,A -85,B 0,C 180,E1 30188.396,E2 30188.396} C_VEL
LIN {X 0,Y 664.435,Z 302.698,A -85,B 0,C 180,E1 30188.01,E2 30188.01} C_VEL
LIN {X 0,Y 666.726,Z 319.035,A -85,B 0,C 180,E1 30187.652,E2 30187.652} C_VEL
LIN {X 0,Y 664.185,Z 578.073,A -85,B 0,C 180,E1 30184.527,E2 30184.527} C_VEL
LIN {X 0,Y 663.137,Z 691.841,A -85,B 0,C 180,E1 30183.175,E2 30183.175} C_VEL
LIN {X 0,Y 662.495,Z 717.649,A -85,B 0,C 180,E1 30182.715,E2 30182.715} C_VEL
LIN {X 0,Y 661.775,Z 739.01,A -85,B 0,C 180,E1 30182.204,E2 30182.204} C_VEL
LIN {X 0,Y 660.812,Z 761.255,A -85,B 0,C 180,E1 30181.519,E2 30181.519} C_VEL
LIN {X 0,Y 659.599,Z 783.335,A -85,B 0,C 180,E1 30180.671,E2 30180.671} C_VEL
LIN {X 0,Y 658.38,Z 805.273,A -85,B 0,C 180,E1 30179.676,E2 30179.676} C_VEL
LIN {X 0,Y 656.935,Z 827.118,A -85,B 0,C 180,E1 30178.5,E2 30178.5} C_VEL
LIN {X 0,Y 655.618,Z 847.65,A -85,B 0,C 180,E1 30177.228,E2 30177.228} C_VEL
LIN {X 0,Y 654.267,Z 867.218,A -85,B 0,C 180,E1 30175.821,E2 30175.821} C_VEL
LIN {X 0,Y 653.067,Z 885.201,A -85,B 0,C 180,E1 30174.357,E2 30174.357} C_VEL
LIN {X 0,Y 651.923,Z 902.603,A -85,B 0,C 180,E1 30172.737,E2 30172.737} C_VEL
LIN {X 0,Y 650.986,Z 917.629,A -85,B 0,C 180,E1 30171.159,E2 30171.159} C_VEL
LIN {X 0,Y 650.064,Z 934.017,A -85,B 0,C 180,E1 30169.192,E2 30169.192} C_VEL
LIN {X 0,Y 649.404,Z 947.155,A -85,B 0,C 180,E1 30167.38,E2 30167.38} C_VEL
LIN {X 0,Y 648.818,Z 960.384,A -85,B 0,C 180,E1 30165.262,E2 30165.262} C_VEL
LIN {X 0,Y 648.459,Z 970.021,A -85,B 0,C 180,E1 30163.464,E2 30163.464} C_VEL
LIN {X 0,Y 648.175,Z 979.834,A -85,B 0,C 180,E1 30161.298,E2 30161.298} C_VEL
LIN {X 0,Y 648.054,Z 986.817,A -85,B 0,C 180,E1 30159.413,E2 30159.413} C_VEL
LIN {X 0,Y 647.946,Z 993.244,A -85,B 0,C 180,E1 30157.27,E2 30157.27} C_VEL
LIN {X 0,Y 647.896,Z 997.656,A -85,B 0,C 180,E1 30155.224,E2 30155.224} C_VEL
LIN {X 0,Y 647.904,Z 1000.463,A -85,B 0,C 180,E1 30153.362,E2 30153.362} C_VEL
LIN {X 0,Y 647.909,Z 1002.215,A -85,B 0,C 180,E1 30151.15,E2 30151.15} C_VEL
LIN {X 0,Y 647.885,Z 1002.328,A -85,B 0,C 180,E1 30149.293,E2 30149.293} C_VEL
LIN {X 0,Y 647.888,Z 1001.225,A -85,B 0,C 180,E1 30147.346,E2 30147.346} C_VEL
LIN {X 0,Y 647.903,Z 998.291,A -85,B 0,C 180,E1 30145.131,E2 30145.131} C_VEL
LIN {X 0,Y 647.937,Z 994.689,A -85,B 0,C 180,E1 30143.354,E2 30143.354} C_VEL
LIN {X 0,Y 647.991,Z 989.202,A -85,B 0,C 180,E1 30141.302,E2 30141.302} C_VEL
LIN {X 0,Y 648.14,Z 981.956,A -85,B 0,C 180,E1 30139.242,E2 30139.242} C_VEL
LIN {X 0,Y 648.361,Z 973.937,A -85,B 0,C 180,E1 30137.35,E2 30137.35} C_VEL
LIN {X 0,Y 648.736,Z 962.864,A -85,B 0,C 180,E1 30135.176,E2 30135.176} C_VEL
LIN {X 0,Y 649.179,Z 951.908,A -85,B 0,C 180,E1 30133.342,E2 30133.342} C_VEL
LIN {X 0,Y 649.881,Z 937.323,A -85,B 0,C 180,E1 30131.242,E2 30131.242} C_VEL
LIN {X 0,Y 650.669,Z 923.308,A -85,B 0,C 180,E1 30129.49,E2 30129.49} C_VEL
LIN {X 0,Y 651.685,Z 906.306,A -85,B 0,C 180,E1 30127.635,E2 30127.635} C_VEL
LIN {X 0,Y 652.725,Z 890.29,A -85,B 0,C 180,E1 30126.098,E2 30126.098} C_VEL
LIN {X 0,Y 654.04,Z 870.36,A -85,B 0,C 180,E1 30124.421,E2 30124.421} C_VEL
LIN {X 0,Y 655.281,Z 852.393,A -85,B 0,C 180,E1 30123.1,E2 30123.1} C_VEL
LIN {X 0,Y 656.73,Z 830.354,A -85,B 0,C 180,E1 30121.688,E2 30121.688} C_VEL
LIN {X 0,Y 657.987,Z 810.743,A -85,B 0,C 180,E1 30120.604,E2 30120.604} C_VEL
LIN {X 0,Y 659.434,Z 786.726,A -85,B 0,C 180,E1 30119.472,E2 30119.472} C_VEL
LIN {X 0,Y 660.465,Z 767.674,A -85,B 0,C 180,E1 30118.716,E2 30118.716} C_VEL
LIN {X 0,Y 661.518,Z 746.017,A -85,B 0,C 180,E1 30117.991,E2 30117.991} C_VEL
LIN {X 0,Y 662.289,Z 722.664,A -85,B 0,C 180,E1 30117.396,E2 30117.396} C_VEL
LIN {X 0,Y 662.833,Z 700.466,A -85,B 0,C 180,E1 30116.978,E2 30116.978} C_VEL
LIN {X 0,Y 663.226,Z 667.583,A -85,B 0,C 180,E1 30116.559,E2 30116.559} C_VEL
LIN {X 0,Y 664.223,Z 431.13,A -85,B 0,C 180,E1 30113.925,E2 30113.925} C_VEL
LIN {X 0,Y 664.615,Z 316.21,A -85,B 0,C 180,E1 30112.595,E2 30112.595} C_VEL
LIN {X 0,Y 662.885,Z 306.048,A -85,B 0,C 180,E1 30112.386,E2 30112.386} C_VEL
LIN {X 0,Y 664.642,Z 271.267,A -85,B 0,C 180,E1 30110.59,E2 30110.59} C_VEL
LIN {X 0,Y 667.165,Z 243.082,A -85,B 0,C 180,E1 30108.991,E2 30108.991} C_VEL
LIN {X 0,Y 663.154,Z 233.195,A -85,B 0,C 180,E1 30107.859,E2 30107.859} C_VEL
LIN {X 0,Y 660.075,Z 226.378,A -85,B 0,C 180,E1 30106.898,E2 30106.898} C_VEL
LIN {X 0,Y 658.312,Z 222.717,A -85,B 0,C 180,E1 30106.284,E2 30106.284} C_VEL
LIN {X 0,Y 656.59,Z 219.08,A -85,B 0,C 180,E1 30105.579,E2 30105.579} C_VEL
LIN {X 0,Y 654.484,Z 214.797,A -85,B 0,C 180,E1 30104.527,E2 30104.527} C_VEL
LIN {X 0,Y 652.478,Z 211.672,A -85,B 0,C 180,E1 30103.16,E2 30103.16} C_VEL
LIN {X 0,Y 652.161,Z 210.241,A -85,B 0,C 180,E1 30102.068,E2 30102.068} C_VEL
LIN {X 0,Y 652.217,Z 210.604,A -85,B 0,C 180,E1 30101.124,E2 30101.124} C_VEL
LIN {X 0,Y 653.16,Z 213.211,A -85,B 0,C 180,E1 30099.782,E2 30099.782} C_VEL
LIN {X 0,Y 654.639,Z 215.367,A -85,B 0,C 180,E1 30098.973,E2 30098.973} C_VEL
LIN {X 0,Y 656.516,Z 219.112,A -85,B 0,C 180,E1 30098.056,E2 30098.056} C_VEL
LIN {X 0,Y 659.162,Z 225.507,A -85,B 0,C 180,E1 30096.92,E2 30096.92} C_VEL
LIN {X 0,Y 662.192,Z 233.136,A -85,B 0,C 180,E1 30095.82,E2 30095.82} C_VEL
LIN {X 0,Y 664.172,Z 238.986,A -85,B 0,C 180,E1 30095.106,E2 30095.106} C_VEL
LIN {X 0,Y 660.624,Z 275.053,A -85,B 0,C 180,E1 30092.604,E2 30092.604} C_VEL
LIN {X 0,Y 657.552,Z 322.58,A -85,B 0,C 180,E1 30089.517,E2 30089.517} C_VEL
LIN {X 0,Y 655.519,Z 368.995,A -85,B 0,C 180,E1 30086.639,E2 30086.639} C_VEL
LIN {X 0,Y 653.654,Z 424.889,A -85,B 0,C 180,E1 30083.293,E2 30083.293} C_VEL
LIN {X 0,Y 653.059,Z 449.561,A -85,B 0,C 180,E1 30081.872,E2 30081.872} C_VEL
LIN {X 0,Y 656.988,Z 483.372,A -85,B 0,C 180,E1 30081.098,E2 30081.098} C_VEL
LIN {X 0,Y 654.028,Z 608.597,A -85,B 0,C 180,E1 30079.304,E2 30079.304} C_VEL
LIN {X 0,Y 652.919,Z 683.38,A -85,B 0,C 180,E1 30078.282,E2 30078.282} C_VEL
LIN {X 0,Y 652.51,Z 703.626,A -85,B 0,C 180,E1 30077.838,E2 30077.838} C_VEL
LIN {X 0,Y 652.068,Z 722.573,A -85,B 0,C 180,E1 30077.261,E2 30077.261} C_VEL
LIN {X 0,Y 651.536,Z 741.817,A -85,B 0,C 180,E1 30076.494,E2 30076.494} C_VEL
LIN {X 0,Y 651.061,Z 758.714,A -85,B 0,C 180,E1 30075.647,E2 30075.647} C_VEL
LIN {X 0,Y 650.555,Z 774.907,A -85,B 0,C 180,E1 30074.654,E2 30074.654} C_VEL
LIN {X 0,Y 650.067,Z 789.577,A -85,B 0,C 180,E1 30073.566,E2 30073.566} C_VEL
LIN {X 0,Y 649.64,Z 802.211,A -85,B 0,C 180,E1 30072.444,E2 30072.444} C_VEL
LIN {X 0,Y 649.249,Z 814.143,A -85,B 0,C 180,E1 30071.179,E2 30071.179} C_VEL
LIN {X 0,Y 648.901,Z 825.187,A -85,B 0,C 180,E1 30069.759,E2 30069.759} C_VEL
LIN {X 0,Y 648.634,Z 834.216,A -85,B 0,C 180,E1 30068.332,E2 30068.332} C_VEL
LIN {X 0,Y 648.438,Z 842.116,A -85,B 0,C 180,E1 30066.759,E2 30066.759} C_VEL
LIN {X 0,Y 648.319,Z 848.304,A -85,B 0,C 180,E1 30065.132,E2 30065.132} C_VEL
LIN {X 0,Y 648.225,Z 852.586,A -85,B 0,C 180,E1 30063.537,E2 30063.537} C_VEL
LIN {X 0,Y 648.176,Z 855.317,A -85,B 0,C 180,E1 30061.856,E2 30061.856} C_VEL
LIN {X 0,Y 648.153,Z 856.294,A -85,B 0,C 180,E1 30060.177,E2 30060.177} C_VEL
LIN {X 0,Y 648.138,Z 855.546,A -85,B 0,C 180,E1 30058.497,E2 30058.497} C_VEL
LIN {X 0,Y 648.156,Z 853.062,A -85,B 0,C 180,E1 30056.816,E2 30056.816} C_VEL
LIN {X 0,Y 648.196,Z 849,A -85,B 0,C 180,E1 30055.209,E2 30055.209} C_VEL
LIN {X 0,Y 648.282,Z 843.29,A -85,B 0,C 180,E1 30053.624,E2 30053.624} C_VEL
LIN {X 0,Y 648.429,Z 835.65,A -85,B 0,C 180,E1 30052.023,E2 30052.023} C_VEL
LIN {X 0,Y 648.665,Z 826.463,A -85,B 0,C 180,E1 30050.506,E2 30050.506} C_VEL
LIN {X 0,Y 648.978,Z 815.776,A -85,B 0,C 180,E1 30049.076,E2 30049.076} C_VEL
LIN {X 0,Y 649.367,Z 803.582,A -85,B 0,C 180,E1 30047.732,E2 30047.732} C_VEL
LIN {X 0,Y 649.833,Z 789.819,A -85,B 0,C 180,E1 30046.474,E2 30046.474} C_VEL
LIN {X 0,Y 650.339,Z 774.993,A -85,B 0,C 180,E1 30045.35,E2 30045.35} C_VEL
LIN {X 0,Y 650.865,Z 759.237,A -85,B 0,C 180,E1 30044.359,E2 30044.359} C_VEL
LIN {X 0,Y 651.383,Z 741.984,A -85,B 0,C 180,E1 30043.472,E2 30043.472} C_VEL
LIN {X 0,Y 651.915,Z 724,A -85,B 0,C 180,E1 30042.735,E2 30042.735} C_VEL
LIN {X 0,Y 652.363,Z 705.072,A -85,B 0,C 180,E1 30042.139,E2 30042.139} C_VEL
LIN {X 0,Y 652.749,Z 685.577,A -85,B 0,C 180,E1 30041.701,E2 30041.701} C_VEL
LIN {X 0,Y 653.055,Z 660.087,A -85,B 0,C 180,E1 30041.347,E2 30041.347} C_VEL
LIN {X 0,Y 654.97,Z 481.489,A -85,B 0,C 180,E1 30039.145,E2 30039.145} C_VEL
LIN {X 0,Y 653.858,Z 472.31,A -85,B 0,C 180,E1 30038.983,E2 30038.983} C_VEL
LIN {X 0,Y 652.368,Z 467.523,A -85,B 0,C 180,E1 30038.844,E2 30038.844} C_VEL
LIN {X 0,Y 648.117,Z 460.613,A -85,B 0,C 180,E1 30038.463,E2 30038.463} C_VEL
LIN {X 0,Y 645.709,Z 455.501,A -85,B 0,C 180,E1 30038.118,E2 30038.118} C_VEL
LIN {X 0,Y 645.421,Z 453.034,A -85,B 0,C 180,E1 30037.965,E2 30037.965} C_VEL
LIN {X 0,Y 646.89,Z 401.363,A -85,B 0,C 180,E1 30034.928,E2 30034.928} C_VEL
LIN {X 0,Y 648.629,Z 348.941,A -85,B 0,C 180,E1 30031.804,E2 30031.804} C_VEL
LIN {X 0,Y 650.482,Z 295.296,A -85,B 0,C 180,E1 30028.553,E2 30028.553} C_VEL
LIN {X 0,Y 652.355,Z 247.523,A -85,B 0,C 180,E1 30025.61,E2 30025.61} C_VEL
LIN {X 0,Y 652.743,Z 236.826,A -85,B 0,C 180,E1 30024.94,E2 30024.94} C_VEL
LIN {X 0,Y 643.253,Z 211.934,A -85,B 0,C 180,E1 30022.737,E2 30022.737} C_VEL
LIN {X 0,Y 640.828,Z 205.41,A -85,B 0,C 180,E1 30022.141,E2 30022.141} C_VEL
LIN {X 0,Y 640.773,Z 205.416,A -85,B 0,C 180,E1 30019.169,E2 30019.169} C_VEL
LIN {X 0,Y 640.8,Z 205.409,A -85,B 0,C 180,E1 30016,E2 30016} C_VEL
LIN {X 0,Y 640.808,Z 205.405,A -85,B 0,C 180,E1 30012.991,E2 30012.991} C_VEL
LIN {X 0,Y 640.791,Z 205.412,A -85,B 0,C 180,E1 30009.85,E2 30009.85} C_VEL
LIN {X 0,Y 640.821,Z 205.644,A -85,B 0,C 180,E1 30008.724,E2 30008.724} C_VEL
LIN {X 0,Y 649.199,Z 226.246,A -85,B 0,C 180,E1 30006.784,E2 30006.784} C_VEL
LIN {X 0,Y 654.391,Z 240.008,A -85,B 0,C 180,E1 30005.418,E2 30005.418} C_VEL
LIN {X 0,Y 653.041,Z 276.512,A -85,B 0,C 180,E1 30002.717,E2 30002.717} C_VEL
LIN {X 0,Y 652.349,Z 308.899,A -85,B 0,C 180,E1 30000.436,E2 30000.436} C_VEL
LIN {X 0,Y 652.483,Z 320.092,A -85,B 0,C 180,E1 29999.716,E2 29999.716} C_VEL
LIN {X 0,Y 653.351,Z 326.024,A -85,B 0,C 180,E1 29999.595,E2 29999.595} C_VEL
LIN {X 0,Y 651.375,Z 465.842,A -85,B 0,C 180,E1 29997.854,E2 29997.854} C_VEL
LIN {X 0,Y 649.238,Z 615.863,A -85,B 0,C 180,E1 29995.915,E2 29995.915} C_VEL
LIN {X 0,Y 648.756,Z 638.263,A -85,B 0,C 180,E1 29995.455,E2 29995.455} C_VEL
LIN {X 0,Y 648.087,Z 660.194,A -85,B 0,C 180,E1 29994.837,E2 29994.837} C_VEL
LIN {X 0,Y 647.338,Z 681.426,A -85,B 0,C 180,E1 29994.065,E2 29994.065} C_VEL
LIN {X 0,Y 646.5,Z 701.268,A -85,B 0,C 180,E1 29993.18,E2 29993.18} C_VEL
LIN {X 0,Y 645.592,Z 720.156,A -85,B 0,C 180,E1 29992.152,E2 29992.152} C_VEL
LIN {X 0,Y 644.604,Z 738.54,A -85,B 0,C 180,E1 29990.963,E2 29990.963} C_VEL
LIN {X 0,Y 643.611,Z 756.559,A -85,B 0,C 180,E1 29989.581,E2 29989.581} C_VEL
LIN {X 0,Y 642.804,Z 770.655,A -85,B 0,C 180,E1 29988.313,E2 29988.313} C_VEL
LIN {X 0,Y 642.12,Z 783.236,A -85,B 0,C 180,E1 29987.023,E2 29987.023} C_VEL
LIN {X 0,Y 641.566,Z 794.393,A -85,B 0,C 180,E1 29985.735,E2 29985.735} C_VEL
LIN {X 0,Y 641.041,Z 806.241,A -85,B 0,C 180,E1 29984.175,E2 29984.175} C_VEL
LIN {X 0,Y 640.558,Z 818.494,A -85,B 0,C 180,E1 29982.257,E2 29982.257} C_VEL
LIN {X 0,Y 640.296,Z 827.228,A -85,B 0,C 180,E1 29980.619,E2 29980.619} C_VEL
LIN {X 0,Y 640.119,Z 834.156,A -85,B 0,C 180,E1 29979.077,E2 29979.077} C_VEL
LIN {X 0,Y 640.003,Z 839.874,A -85,B 0,C 180,E1 29977.541,E2 29977.541} C_VEL
LIN {X 0,Y 639.952,Z 844.477,A -85,B 0,C 180,E1 29976.009,E2 29976.009} C_VEL
LIN {X 0,Y 639.927,Z 848.355,A -85,B 0,C 180,E1 29974.301,E2 29974.301} C_VEL
LIN {X 0,Y 639.912,Z 851.284,A -85,B 0,C 180,E1 29972.328,E2 29972.328} C_VEL
LIN {X 0,Y 639.904,Z 852.406,A -85,B 0,C 180,E1 29970.269,E2 29970.269} C_VEL
LIN {X 0,Y 639.898,Z 851.993,A -85,B 0,C 180,E1 29968.567,E2 29968.567} C_VEL
LIN {X 0,Y 639.902,Z 850.469,A -85,B 0,C 180,E1 29966.955,E2 29966.955} C_VEL
LIN {X 0,Y 639.921,Z 847.819,A -85,B 0,C 180,E1 29965.34,E2 29965.34} C_VEL
LIN {X 0,Y 639.963,Z 843.997,A -85,B 0,C 180,E1 29963.721,E2 29963.721} C_VEL
LIN {X 0,Y 640.025,Z 838.659,A -85,B 0,C 180,E1 29962.008,E2 29962.008} C_VEL
LIN {X 0,Y 640.203,Z 830.73,A -85,B 0,C 180,E1 29960.017,E2 29960.017} C_VEL
LIN {X 0,Y 640.459,Z 821.549,A -85,B 0,C 180,E1 29958.199,E2 29958.199} C_VEL
LIN {X 0,Y 640.761,Z 812.893,A -85,B 0,C 180,E1 29956.739,E2 29956.739} C_VEL
LIN {X 0,Y 641.147,Z 803.547,A -85,B 0,C 180,E1 29955.366,E2 29955.366} C_VEL
LIN {X 0,Y 641.609,Z 793.434,A -85,B 0,C 180,E1 29954.059,E2 29954.059} C_VEL
LIN {X 0,Y 642.168,Z 782.351,A -85,B 0,C 180,E1 29952.792,E2 29952.792} C_VEL
LIN {X 0,Y 642.858,Z 769.665,A -85,B 0,C 180,E1 29951.5,E2 29951.5} C_VEL
LIN {X 0,Y 643.734,Z 754.551,A -85,B 0,C 180,E1 29950.16,E2 29950.16} C_VEL
LIN {X 0,Y 644.709,Z 736.664,A -85,B 0,C 180,E1 29948.816,E2 29948.816} C_VEL
LIN {X 0,Y 645.707,Z 717.565,A -85,B 0,C 180,E1 29947.608,E2 29947.608} C_VEL
LIN {X 0,Y 646.617,Z 698.841,A -85,B 0,C 180,E1 29946.612,E2 29946.612} C_VEL
LIN {X 0,Y 647.437,Z 678.959,A -85,B 0,C 180,E1 29945.745,E2 29945.745} C_VEL
LIN {X 0,Y 648.111,Z 659.134,A -85,B 0,C 180,E1 29945.042,E2 29945.042} C_VEL
LIN {X 0,Y 648.75,Z 638.223,A -85,B 0,C 180,E1 29944.456,E2 29944.456} C_VEL
LIN {X 0,Y 649.218,Z 616.481,A -85,B 0,C 180,E1 29944.006,E2 29944.006} C_VEL
LIN {X 0,Y 649.909,Z 565.175,A -85,B 0,C 180,E1 29943.33,E2 29943.33} C_VEL
LIN {X 0,Y 652.937,Z 359.404,A -85,B 0,C 180,E1 29940.718,E2 29940.718} C_VEL
LIN {X 0,Y 653.179,Z 323.688,A -85,B 0,C 180,E1 29940.276,E2 29940.276} C_VEL
LIN {X 0,Y 652.385,Z 319.37,A -85,B 0,C 180,E1 29940.169,E2 29940.169} C_VEL
LIN {X 0,Y 652.738,Z 286.092,A -85,B 0,C 180,E1 29937.89,E2 29937.89} C_VEL
LIN {X 0,Y 654.227,Z 245.943,A -85,B 0,C 180,E1 29934.924,E2 29934.924} C_VEL
LIN {X 0,Y 654.341,Z 239.728,A -85,B 0,C 180,E1 29934.46,E2 29934.46} C_VEL
LIN {X 0,Y 647.416,Z 221.801,A -85,B 0,C 180,E1 29932.692,E2 29932.692} C_VEL
LIN {X 0,Y 640.89,Z 205.935,A -85,B 0,C 180,E1 29931.2,E2 29931.2} C_VEL
LIN {X 0,Y 640.804,Z 205.413,A -85,B 0,C 180,E1 29931.135,E2 29931.135} C_VEL
LIN {X 0,Y 640.827,Z 205.408,A -85,B 0,C 180,E1 29928.097,E2 29928.097} C_VEL
LIN {X 0,Y 640.803,Z 205.411,A -85,B 0,C 180,E1 29924.979,E2 29924.979} C_VEL
LIN {X 0,Y 640.822,Z 205.409,A -85,B 0,C 180,E1 29921.899,E2 29921.899} C_VEL
LIN {X 0,Y 640.806,Z 205.408,A -85,B 0,C 180,E1 29918.849,E2 29918.849} C_VEL
LIN {X 0,Y 640.82,Z 205.406,A -85,B 0,C 180,E1 29915.77,E2 29915.77} C_VEL
LIN {X 0,Y 640.81,Z 205.397,A -85,B 0,C 180,E1 29912.676,E2 29912.676} C_VEL
LIN {X 0,Y 640.823,Z 205.397,A -85,B 0,C 180,E1 29909.542,E2 29909.542} C_VEL
LIN {X 0,Y 640.823,Z 205.406,A -85,B 0,C 180,E1 29906.404,E2 29906.404} C_VEL
LIN {X 0,Y 640.826,Z 205.386,A -85,B 0,C 180,E1 29903.154,E2 29903.154} C_VEL
LIN {X 0,Y 640.818,Z 205.401,A -85,B 0,C 180,E1 29899.981,E2 29899.981} C_VEL
LIN {X 0,Y 640.817,Z 205.393,A -85,B 0,C 180,E1 29896.871,E2 29896.871} C_VEL
LIN {X 0,Y 640.81,Z 205.397,A -85,B 0,C 180,E1 29893.812,E2 29893.812} C_VEL
LIN {X 0,Y 640.818,Z 205.395,A -85,B 0,C 180,E1 29890.701,E2 29890.701} C_VEL
LIN {X 0,Y 640.805,Z 205.398,A -85,B 0,C 180,E1 29887.622,E2 29887.622} C_VEL
LIN {X 0,Y 640.819,Z 205.394,A -85,B 0,C 180,E1 29884.564,E2 29884.564} C_VEL
LIN {X 0,Y 640.803,Z 205.401,A -85,B 0,C 180,E1 29881.52,E2 29881.52} C_VEL
LIN {X 0,Y 640.822,Z 205.388,A -85,B 0,C 180,E1 29878.48,E2 29878.48} C_VEL
LIN {X 0,Y 640.801,Z 205.403,A -85,B 0,C 180,E1 29875.436,E2 29875.436} C_VEL
LIN {X 0,Y 640.826,Z 205.388,A -85,B 0,C 180,E1 29872.288,E2 29872.288} C_VEL
LIN {X 0,Y 640.805,Z 205.403,A -85,B 0,C 180,E1 29869.208,E2 29869.208} C_VEL
LIN {X 0,Y 640.82,Z 205.409,A -85,B 0,C 180,E1 29866.004,E2 29866.004} C_VEL
LIN {X 0,Y 640.826,Z 205.403,A -85,B 0,C 180,E1 29862.848,E2 29862.848} C_VEL
LIN {X 0,Y 640.797,Z 205.408,A -85,B 0,C 180,E1 29859.684,E2 29859.684} C_VEL
LIN {X 0,Y 640.834,Z 205.404,A -85,B 0,C 180,E1 29856.652,E2 29856.652} C_VEL
LIN {X 0,Y 640.792,Z 205.405,A -85,B 0,C 180,E1 29853.594,E2 29853.594} C_VEL
LIN {X 0,Y 640.834,Z 205.402,A -85,B 0,C 180,E1 29850.534,E2 29850.534} C_VEL
LIN {X 0,Y 640.786,Z 205.411,A -85,B 0,C 180,E1 29847.535,E2 29847.535} C_VEL
LIN {X 0,Y 640.831,Z 205.406,A -85,B 0,C 180,E1 29844.519,E2 29844.519} C_VEL
LIN {X 0,Y 640.78,Z 205.411,A -85,B 0,C 180,E1 29841.423,E2 29841.423} C_VEL
LIN {X 0,Y 640.835,Z 205.403,A -85,B 0,C 180,E1 29838.461,E2 29838.461} C_VEL
LIN {X 0,Y 640.776,Z 205.412,A -85,B 0,C 180,E1 29835.362,E2 29835.362} C_VEL
LIN {X 0,Y 642.076,Z 208.877,A -85,B 0,C 180,E1 29835.008,E2 29835.008} C_VEL
LIN {X 0,Y 643.369,Z 211.316,A -85,B 0,C 180,E1 29834.745,E2 29834.745} C_VEL
LIN {X 0,Y 653.762,Z 232.116,A -85,B 0,C 180,E1 29832.637,E2 29832.637} C_VEL
LIN {X 0,Y 660.528,Z 246.496,A -85,B 0,C 180,E1 29831.296,E2 29831.296} C_VEL
LIN {X 0,Y 657.722,Z 303.299,A -85,B 0,C 180,E1 29828.406,E2 29828.406} C_VEL
LIN {X 0,Y 660.087,Z 320.461,A -85,B 0,C 180,E1 29828.025,E2 29828.025} C_VEL
LIN {X 0,Y 657.225,Z 576.361,A -85,B 0,C 180,E1 29824.889,E2 29824.889} C_VEL
LIN {X 0,Y 656.033,Z 691.701,A -85,B 0,C 180,E1 29823.499,E2 29823.499} C_VEL
LIN {X 0,Y 655.355,Z 717.299,A -85,B 0,C 180,E1 29823.039,E2 29823.039} C_VEL
LIN {X 0,Y 654.581,Z 738.856,A -85,B 0,C 180,E1 29822.518,E2 29822.518} C_VEL
LIN {X 0,Y 653.482,Z 764.441,A -85,B 0,C 180,E1 29821.73,E2 29821.73} C_VEL
LIN {X 0,Y 652.452,Z 785.308,A -85,B 0,C 180,E1 29820.941,E2 29820.941} C_VEL
LIN {X 0,Y 651.303,Z 805.277,A -85,B 0,C 180,E1 29820.032,E2 29820.032} C_VEL
LIN {X 0,Y 649.76,Z 827.032,A -85,B 0,C 180,E1 29818.849,E2 29818.849} C_VEL
LIN {X 0,Y 648.313,Z 847.653,A -85,B 0,C 180,E1 29817.561,E2 29817.561} C_VEL
LIN {X 0,Y 646.864,Z 867.215,A -85,B 0,C 180,E1 29816.138,E2 29816.138} C_VEL
LIN {X 0,Y 645.559,Z 885.061,A -85,B 0,C 180,E1 29814.672,E2 29814.672} C_VEL
LIN {X 0,Y 644.311,Z 902.602,A -85,B 0,C 180,E1 29813.021,E2 29813.021} C_VEL
LIN {X 0,Y 643.278,Z 917.865,A -85,B 0,C 180,E1 29811.398,E2 29811.398} C_VEL
LIN {X 0,Y 642.3,Z 933.819,A -85,B 0,C 180,E1 29809.459,E2 29809.459} C_VEL
LIN {X 0,Y 641.574,Z 946.518,A -85,B 0,C 180,E1 29807.692,E2 29807.692} C_VEL
LIN {X 0,Y 640.936,Z 959.769,A -85,B 0,C 180,E1 29805.565,E2 29805.565} C_VEL
LIN {X 0,Y 640.537,Z 969.561,A -85,B 0,C 180,E1 29803.726,E2 29803.726} C_VEL
LIN {X 0,Y 640.242,Z 979.124,A -85,B 0,C 180,E1 29801.623,E2 29801.623} C_VEL
LIN {X 0,Y 640.069,Z 986.514,A -85,B 0,C 180,E1 29799.622,E2 29799.622} C_VEL
LIN {X 0,Y 639.945,Z 992.762,A -85,B 0,C 180,E1 29797.542,E2 29797.542} C_VEL
LIN {X 0,Y 639.901,Z 997.496,A -85,B 0,C 180,E1 29795.38,E2 29795.38} C_VEL
LIN {X 0,Y 639.911,Z 1000.351,A -85,B 0,C 180,E1 29793.494,E2 29793.494} C_VEL
LIN {X 0,Y 639.908,Z 1002.192,A -85,B 0,C 180,E1 29791.253,E2 29791.253} C_VEL
LIN {X 0,Y 639.885,Z 1002.328,A -85,B 0,C 180,E1 29789.284,E2 29789.284} C_VEL
LIN {X 0,Y 639.887,Z 1001.225,A -85,B 0,C 180,E1 29787.313,E2 29787.313} C_VEL
LIN {X 0,Y 639.901,Z 998.292,A -85,B 0,C 180,E1 29785.07,E2 29785.07} C_VEL
LIN {X 0,Y 639.944,Z 994.689,A -85,B 0,C 180,E1 29783.27,E2 29783.27} C_VEL
LIN {X 0,Y 640.007,Z 988.934,A -85,B 0,C 180,E1 29781.102,E2 29781.102} C_VEL
LIN {X 0,Y 640.164,Z 981.603,A -85,B 0,C 180,E1 29779.015,E2 29779.015} C_VEL
LIN {X 0,Y 640.421,Z 973.53,A -85,B 0,C 180,E1 29777.099,E2 29777.099} C_VEL
LIN {X 0,Y 640.82,Z 962.834,A -85,B 0,C 180,E1 29774.983,E2 29774.983} C_VEL
LIN {X 0,Y 641.311,Z 951.973,A -85,B 0,C 180,E1 29773.142,E2 29773.142} C_VEL
LIN {X 0,Y 642.078,Z 937.321,A -85,B 0,C 180,E1 29771.006,E2 29771.006} C_VEL
LIN {X 0,Y 642.89,Z 924.078,A -85,B 0,C 180,E1 29769.326,E2 29769.326} C_VEL
LIN {X 0,Y 643.993,Z 907.23,A -85,B 0,C 180,E1 29767.449,E2 29767.449} C_VEL
LIN {X 0,Y 645.091,Z 891.542,A -85,B 0,C 180,E1 29765.917,E2 29765.917} C_VEL
LIN {X 0,Y 646.455,Z 872.685,A -85,B 0,C 180,E1 29764.287,E2 29764.287} C_VEL
LIN {X 0,Y 647.801,Z 854.392,A -85,B 0,C 180,E1 29762.913,E2 29762.913} C_VEL
LIN {X 0,Y 649.326,Z 833.594,A -85,B 0,C 180,E1 29761.537,E2 29761.537} C_VEL
LIN {X 0,Y 650.699,Z 813.328,A -85,B 0,C 180,E1 29760.388,E2 29760.388} C_VEL
LIN {X 0,Y 652.091,Z 792.534,A -85,B 0,C 180,E1 29759.365,E2 29759.365} C_VEL
LIN {X 0,Y 653.112,Z 771.457,A -85,B 0,C 180,E1 29758.529,E2 29758.529} C_VEL
LIN {X 0,Y 653.982,Z 749.69,A -85,B 0,C 180,E1 29757.827,E2 29757.827} C_VEL
LIN {X 0,Y 654.804,Z 724.006,A -85,B 0,C 180,E1 29757.166,E2 29757.166} C_VEL
LIN {X 0,Y 655.401,Z 700.977,A -85,B 0,C 180,E1 29756.725,E2 29756.725} C_VEL
LIN {X 0,Y 655.819,Z 668.673,A -85,B 0,C 180,E1 29756.305,E2 29756.305} C_VEL
LIN {X 0,Y 656.905,Z 438,A -85,B 0,C 180,E1 29753.714,E2 29753.714} C_VEL
LIN {X 0,Y 657.494,Z 317.486,A -85,B 0,C 180,E1 29752.292,E2 29752.292} C_VEL
LIN {X 0,Y 655.903,Z 308.074,A -85,B 0,C 180,E1 29752.095,E2 29752.095} C_VEL
LIN {X 0,Y 657.908,Z 274.941,A -85,B 0,C 180,E1 29750.333,E2 29750.333} C_VEL
LIN {X 0,Y 660.829,Z 246.988,A -85,B 0,C 180,E1 29748.694,E2 29748.694} C_VEL
LIN {X 0,Y 657.133,Z 237.55,A -85,B 0,C 180,E1 29747.559,E2 29747.559} C_VEL
LIN {X 0,Y 653.714,Z 229.544,A -85,B 0,C 180,E1 29746.343,E2 29746.343} C_VEL
LIN {X 0,Y 651.418,Z 224.985,A -85,B 0,C 180,E1 29745.416,E2 29745.416} C_VEL
LIN {X 0,Y 649.639,Z 221.116,A -85,B 0,C 180,E1 29744.425,E2 29744.425} C_VEL
LIN {X 0,Y 647.858,Z 218.188,A -85,B 0,C 180,E1 29743.112,E2 29743.112} C_VEL
LIN {X 0,Y 647.588,Z 216.77,A -85,B 0,C 180,E1 29741.956,E2 29741.956} C_VEL
LIN {X 0,Y 647.605,Z 217.408,A -85,B 0,C 180,E1 29740.974,E2 29740.974} C_VEL
LIN {X 0,Y 648.783,Z 220.148,A -85,B 0,C 180,E1 29739.593,E2 29739.593} C_VEL
LIN {X 0,Y 649.676,Z 221.608,A -85,B 0,C 180,E1 29739.069,E2 29739.069} C_VEL
LIN {X 0,Y 651.664,Z 226.181,A -85,B 0,C 180,E1 29737.973,E2 29737.973} C_VEL
LIN {X 0,Y 654.089,Z 231.929,A -85,B 0,C 180,E1 29736.918,E2 29736.918} C_VEL
LIN {X 0,Y 657.229,Z 240.749,A -85,B 0,C 180,E1 29735.667,E2 29735.667} C_VEL
LIN {X 0,Y 657.877,Z 243.083,A -85,B 0,C 180,E1 29735.385,E2 29735.385} C_VEL
LIN {X 0,Y 654.022,Z 277.586,A -85,B 0,C 180,E1 29732.93,E2 29732.93} C_VEL
LIN {X 0,Y 650.667,Z 322.883,A -85,B 0,C 180,E1 29729.922,E2 29729.922} C_VEL
LIN {X 0,Y 648.399,Z 368.098,A -85,B 0,C 180,E1 29727.06,E2 29727.06} C_VEL
LIN {X 0,Y 646.387,Z 421.369,A -85,B 0,C 180,E1 29723.812,E2 29723.812} C_VEL
LIN {X 0,Y 645.642,Z 446.78,A -85,B 0,C 180,E1 29722.319,E2 29722.319} C_VEL
LIN {X 0,Y 649.975,Z 484.177,A -85,B 0,C 180,E1 29721.43,E2 29721.43} C_VEL
LIN {X 0,Y 646.851,Z 599.918,A -85,B 0,C 180,E1 29719.706,E2 29719.706} C_VEL
LIN {X 0,Y 645.385,Z 683.668,A -85,B 0,C 180,E1 29718.518,E2 29718.518} C_VEL
LIN {X 0,Y 644.939,Z 704.063,A -85,B 0,C 180,E1 29718.064,E2 29718.064} C_VEL
LIN {X 0,Y 644.459,Z 723.235,A -85,B 0,C 180,E1 29717.471,E2 29717.471} C_VEL
LIN {X 0,Y 643.922,Z 741.453,A -85,B 0,C 180,E1 29716.741,E2 29716.741} C_VEL
LIN {X 0,Y 643.38,Z 759.262,A -85,B 0,C 180,E1 29715.845,E2 29715.845} C_VEL
LIN {X 0,Y 642.836,Z 775.536,A -85,B 0,C 180,E1 29714.839,E2 29714.839} C_VEL
LIN {X 0,Y 642.318,Z 790.242,A -85,B 0,C 180,E1 29713.742,E2 29713.742} C_VEL
LIN {X 0,Y 641.856,Z 803.053,A -85,B 0,C 180,E1 29712.597,E2 29712.597} C_VEL
LIN {X 0,Y 641.438,Z 814.956,A -85,B 0,C 180,E1 29711.327,E2 29711.327} C_VEL
LIN {X 0,Y 641.059,Z 826.152,A -85,B 0,C 180,E1 29709.879,E2 29709.879} C_VEL
LIN {X 0,Y 640.758,Z 835.587,A -85,B 0,C 180,E1 29708.371,E2 29708.371} C_VEL
LIN {X 0,Y 640.548,Z 843.291,A -85,B 0,C 180,E1 29706.813,E2 29706.813} C_VEL
LIN {X 0,Y 640.415,Z 849.369,A -85,B 0,C 180,E1 29705.196,E2 29705.196} C_VEL
LIN {X 0,Y 640.309,Z 853.658,A -85,B 0,C 180,E1 29703.581,E2 29703.581} C_VEL
LIN {X 0,Y 640.251,Z 856.386,A -85,B 0,C 180,E1 29701.879,E2 29701.879} C_VEL
LIN {X 0,Y 640.222,Z 857.342,A -85,B 0,C 180,E1 29700.179,E2 29700.179} C_VEL
LIN {X 0,Y 640.204,Z 856.56,A -85,B 0,C 180,E1 29698.479,E2 29698.479} C_VEL
LIN {X 0,Y 640.223,Z 854.029,A -85,B 0,C 180,E1 29696.777,E2 29696.777} C_VEL
LIN {X 0,Y 640.273,Z 849.687,A -85,B 0,C 180,E1 29695.073,E2 29695.073} C_VEL
LIN {X 0,Y 640.369,Z 843.779,A -85,B 0,C 180,E1 29693.455,E2 29693.455} C_VEL
LIN {X 0,Y 640.542,Z 835.96,A -85,B 0,C 180,E1 29691.833,E2 29691.833} C_VEL
LIN {X 0,Y 640.802,Z 826.573,A -85,B 0,C 180,E1 29690.298,E2 29690.298} C_VEL
LIN {X 0,Y 641.144,Z 815.658,A -85,B 0,C 180,E1 29688.85,E2 29688.85} C_VEL
LIN {X 0,Y 641.566,Z 803.212,A -85,B 0,C 180,E1 29687.489,E2 29687.489} C_VEL
LIN {X 0,Y 642.071,Z 789.175,A -85,B 0,C 180,E1 29686.216,E2 29686.216} C_VEL
LIN {X 0,Y 642.627,Z 773.942,A -85,B 0,C 180,E1 29685.07,E2 29685.07} C_VEL
LIN {X 0,Y 643.188,Z 757.942,A -85,B 0,C 180,E1 29684.075,E2 29684.075} C_VEL
LIN {X 0,Y 643.745,Z 740.91,A -85,B 0,C 180,E1 29683.208,E2 29683.208} C_VEL
LIN {X 0,Y 644.306,Z 722.97,A -85,B 0,C 180,E1 29682.478,E2 29682.478} C_VEL
LIN {X 0,Y 644.804,Z 703.329,A -85,B 0,C 180,E1 29681.868,E2 29681.868} C_VEL
LIN {X 0,Y 645.21,Z 683.617,A -85,B 0,C 180,E1 29681.436,E2 29681.436} C_VEL
LIN {X 0,Y 645.584,Z 652.222,A -85,B 0,C 180,E1 29681.013,E2 29681.013} C_VEL
LIN {X 0,Y 647.544,Z 481.946,A -85,B 0,C 180,E1 29678.87,E2 29678.87} C_VEL
LIN {X 0,Y 645.194,Z 462.193,A -85,B 0,C 180,E1 29678.499,E2 29678.499} C_VEL
LIN {X 0,Y 645.421,Z 453.034,A -85,B 0,C 180,E1 29677.965,E2 29677.965} C_VEL
LIN {X 0,Y 644.647,Z 446.758,A -85,B 0,C 180,E1 29677.565,E2 29677.565} C_VEL
LIN {X 0,Y 639.241,Z 430.811,A -85,B 0,C 180,E1 29676.406,E2 29676.406} C_VEL
LIN {X 0,Y 638.723,Z 425.411,A -85,B 0,C 180,E1 29676.058,E2 29676.058} C_VEL
LIN {X 0,Y 640.513,Z 370.69,A -85,B 0,C 180,E1 29672.781,E2 29672.781} C_VEL
LIN {X 0,Y 642.235,Z 323.438,A -85,B 0,C 180,E1 29669.913,E2 29669.913} C_VEL
LIN {X 0,Y 644.421,Z 269.602,A -85,B 0,C 180,E1 29666.592,E2 29666.592} C_VEL
LIN {X 0,Y 645.57,Z 239.683,A -85,B 0,C 180,E1 29664.709,E2 29664.709} C_VEL
LIN {X 0,Y 635.215,Z 212.676,A -85,B 0,C 180,E1 29662.278,E2 29662.278} C_VEL
LIN {X 0,Y 632.843,Z 206.4,A -85,B 0,C 180,E1 29661.673,E2 29661.673} C_VEL
LIN {X 0,Y 632.898,Z 206.394,A -85,B 0,C 180,E1 29658.628,E2 29658.628} C_VEL
LIN {X 0,Y 632.88,Z 206.397,A -85,B 0,C 180,E1 29655.442,E2 29655.442} C_VEL
LIN {X 0,Y 632.893,Z 206.394,A -85,B 0,C 180,E1 29652.301,E2 29652.301} C_VEL
LIN {X 0,Y 632.82,Z 206.401,A -85,B 0,C 180,E1 29649.317,E2 29649.317} C_VEL
LIN {X 0,Y 632.849,Z 206.609,A -85,B 0,C 180,E1 29649.225,E2 29649.225} C_VEL
LIN {X 0,Y 633.955,Z 209.607,A -85,B 0,C 180,E1 29648.961,E2 29648.961} C_VEL
LIN {X 0,Y 641.581,Z 227.74,A -85,B 0,C 180,E1 29647.207,E2 29647.207} C_VEL
LIN {X 0,Y 647.552,Z 243.595,A -85,B 0,C 180,E1 29645.635,E2 29645.635} C_VEL
LIN {X 0,Y 646.093,Z 282.724,A -85,B 0,C 180,E1 29642.744,E2 29642.744} C_VEL
LIN {X 0,Y 645.582,Z 313.879,A -85,B 0,C 180,E1 29640.578,E2 29640.578} C_VEL
LIN {X 0,Y 645.792,Z 322.606,A -85,B 0,C 180,E1 29640.034,E2 29640.034} C_VEL
LIN {X 0,Y 646.431,Z 327.594,A -85,B 0,C 180,E1 29639.936,E2 29639.936} C_VEL
LIN {X 0,Y 644.515,Z 453.18,A -85,B 0,C 180,E1 29638.351,E2 29638.351} C_VEL
LIN {X 0,Y 641.737,Z 617.227,A -85,B 0,C 180,E1 29636.149,E2 29636.149} C_VEL
LIN {X 0,Y 641.238,Z 639.138,A -85,B 0,C 180,E1 29635.686,E2 29635.686} C_VEL
LIN {X 0,Y 640.554,Z 660.587,A -85,B 0,C 180,E1 29635.075,E2 29635.075} C_VEL
LIN {X 0,Y 639.803,Z 681.266,A -85,B 0,C 180,E1 29634.323,E2 29634.323} C_VEL
LIN {X 0,Y 638.923,Z 701.378,A -85,B 0,C 180,E1 29633.422,E2 29633.422} C_VEL
LIN {X 0,Y 637.947,Z 721.125,A -85,B 0,C 180,E1 29632.344,E2 29632.344} C_VEL
LIN {X 0,Y 636.947,Z 739.263,A -85,B 0,C 180,E1 29631.165,E2 29631.165} C_VEL
LIN {X 0,Y 636.039,Z 755.438,A -85,B 0,C 180,E1 29629.932,E2 29629.932} C_VEL
LIN {X 0,Y 635.112,Z 770.997,A -85,B 0,C 180,E1 29628.543,E2 29628.543} C_VEL
LIN {X 0,Y 634.324,Z 784.425,A -85,B 0,C 180,E1 29627.144,E2 29627.144} C_VEL
LIN {X 0,Y 633.571,Z 798.306,A -85,B 0,C 180,E1 29625.469,E2 29625.469} C_VEL
LIN {X 0,Y 632.925,Z 811.14,A -85,B 0,C 180,E1 29623.615,E2 29623.615} C_VEL
LIN {X 0,Y 632.559,Z 820.024,A -85,B 0,C 180,E1 29622.136,E2 29622.136} C_VEL
LIN {X 0,Y 632.32,Z 827.662,A -85,B 0,C 180,E1 29620.662,E2 29620.662} C_VEL
LIN {X 0,Y 632.131,Z 834.521,A -85,B 0,C 180,E1 29619.101,E2 29619.101} C_VEL
LIN {X 0,Y 632.009,Z 840.177,A -85,B 0,C 180,E1 29617.546,E2 29617.546} C_VEL
LIN {X 0,Y 631.947,Z 844.954,A -85,B 0,C 180,E1 29615.903,E2 29615.903} C_VEL
LIN {X 0,Y 631.923,Z 849.065,A -85,B 0,C 180,E1 29613.992,E2 29613.992} C_VEL
LIN {X 0,Y 631.916,Z 851.634,A -85,B 0,C 180,E1 29611.904,E2 29611.904} C_VEL
LIN {X 0,Y 631.907,Z 852.399,A -85,B 0,C 180,E1 29610.181,E2 29610.181} C_VEL
LIN {X 0,Y 631.898,Z 851.988,A -85,B 0,C 180,E1 29608.549,E2 29608.549} C_VEL
LIN {X 0,Y 631.903,Z 850.582,A -85,B 0,C 180,E1 29607.007,E2 29607.007} C_VEL
LIN {X 0,Y 631.922,Z 847.99,A -85,B 0,C 180,E1 29605.371,E2 29605.371} C_VEL
LIN {X 0,Y 631.965,Z 844.23,A -85,B 0,C 180,E1 29603.733,E2 29603.733} C_VEL
LIN {X 0,Y 632.015,Z 839.565,A -85,B 0,C 180,E1 29602.18,E2 29602.18} C_VEL
LIN {X 0,Y 632.143,Z 833.775,A -85,B 0,C 180,E1 29600.624,E2 29600.624} C_VEL
LIN {X 0,Y 632.353,Z 826.338,A -85,B 0,C 180,E1 29598.97,E2 29598.97} C_VEL
LIN {X 0,Y 632.74,Z 815.819,A -85,B 0,C 180,E1 29597.033,E2 29597.033} C_VEL
LIN {X 0,Y 633.206,Z 804.873,A -85,B 0,C 180,E1 29595.365,E2 29595.365} C_VEL
LIN {X 0,Y 633.777,Z 794.037,A -85,B 0,C 180,E1 29593.905,E2 29593.905} C_VEL
LIN {X 0,Y 634.431,Z 782.7,A -85,B 0,C 180,E1 29592.576,E2 29592.576} C_VEL
LIN {X 0,Y 635.302,Z 767.838,A -85,B 0,C 180,E1 29591.069,E2 29591.069} C_VEL
LIN {X 0,Y 636.28,Z 751.126,A -85,B 0,C 180,E1 29589.63,E2 29589.63} C_VEL
LIN {X 0,Y 637.196,Z 735.149,A -85,B 0,C 180,E1 29588.457,E2 29588.457} C_VEL
LIN {X 0,Y 638.108,Z 717.554,A -85,B 0,C 180,E1 29587.361,E2 29587.361} C_VEL
LIN {X 0,Y 639.057,Z 698.199,A -85,B 0,C 180,E1 29586.339,E2 29586.339} C_VEL
LIN {X 0,Y 639.905,Z 678.909,A -85,B 0,C 180,E1 29585.49,E2 29585.49} C_VEL
LIN {X 0,Y 640.648,Z 658.096,A -85,B 0,C 180,E1 29584.755,E2 29584.755} C_VEL
LIN {X 0,Y 641.299,Z 636.268,A -85,B 0,C 180,E1 29584.155,E2 29584.155} C_VEL
LIN {X 0,Y 641.783,Z 614.493,A -85,B 0,C 180,E1 29583.72,E2 29583.72} C_VEL
LIN {X 0,Y 645.543,Z 392.365,A -85,B 0,C 180,E1 29580.775,E2 29580.775} C_VEL
LIN {X 0,Y 646.257,Z 325.008,A -85,B 0,C 180,E1 29579.931,E2 29579.931} C_VEL
LIN {X 0,Y 645.682,Z 321.596,A -85,B 0,C 180,E1 29579.834,E2 29579.834} C_VEL
LIN {X 0,Y 645.872,Z 291.858,A -85,B 0,C 180,E1 29577.822,E2 29577.822} C_VEL
LIN {X 0,Y 647.35,Z 249.543,A -85,B 0,C 180,E1 29574.713,E2 29574.713} C_VEL
LIN {X 0,Y 647.501,Z 243.241,A -85,B 0,C 180,E1 29574.243,E2 29574.243} C_VEL
LIN {X 0,Y 640.016,Z 223.753,A -85,B 0,C 180,E1 29572.308,E2 29572.308} C_VEL
LIN {X 0,Y 633.801,Z 209.288,A -85,B 0,C 180,E1 29570.913,E2 29570.913} C_VEL
LIN {X 0,Y 632.869,Z 206.401,A -85,B 0,C 180,E1 29570.644,E2 29570.644} C_VEL
LIN {X 0,Y 632.883,Z 206.396,A -85,B 0,C 180,E1 29567.412,E2 29567.412} C_VEL
LIN {X 0,Y 632.889,Z 206.394,A -85,B 0,C 180,E1 29564.292,E2 29564.292} C_VEL
LIN {X 0,Y 632.87,Z 206.396,A -85,B 0,C 180,E1 29561.091,E2 29561.091} C_VEL
LIN {X 0,Y 632.884,Z 206.393,A -85,B 0,C 180,E1 29558.036,E2 29558.036} C_VEL
LIN {X 0,Y 632.87,Z 206.395,A -85,B 0,C 180,E1 29554.885,E2 29554.885} C_VEL
LIN {X 0,Y 632.88,Z 206.394,A -85,B 0,C 180,E1 29551.79,E2 29551.79} C_VEL
LIN {X 0,Y 632.872,Z 206.386,A -85,B 0,C 180,E1 29548.734,E2 29548.734} C_VEL
LIN {X 0,Y 632.879,Z 206.391,A -85,B 0,C 180,E1 29545.652,E2 29545.652} C_VEL
LIN {X 0,Y 632.88,Z 206.382,A -85,B 0,C 180,E1 29542.479,E2 29542.479} C_VEL
LIN {X 0,Y 632.888,Z 206.382,A -85,B 0,C 180,E1 29539.281,E2 29539.281} C_VEL
LIN {X 0,Y 632.883,Z 206.396,A -85,B 0,C 180,E1 29536.05,E2 29536.05} C_VEL
LIN {X 0,Y 632.882,Z 206.381,A -85,B 0,C 180,E1 29532.89,E2 29532.89} C_VEL
LIN {X 0,Y 632.871,Z 206.396,A -85,B 0,C 180,E1 29529.825,E2 29529.825} C_VEL
LIN {X 0,Y 632.881,Z 206.384,A -85,B 0,C 180,E1 29526.714,E2 29526.714} C_VEL
LIN {X 0,Y 632.866,Z 206.395,A -85,B 0,C 180,E1 29523.623,E2 29523.623} C_VEL
LIN {X 0,Y 632.882,Z 206.387,A -85,B 0,C 180,E1 29520.543,E2 29520.543} C_VEL
LIN {X 0,Y 632.863,Z 206.392,A -85,B 0,C 180,E1 29517.464,E2 29517.464} C_VEL
LIN {X 0,Y 632.888,Z 206.386,A -85,B 0,C 180,E1 29514.288,E2 29514.288} C_VEL
LIN {X 0,Y 632.869,Z 206.387,A -85,B 0,C 180,E1 29511.184,E2 29511.184} C_VEL
LIN {X 0,Y 632.875,Z 206.399,A -85,B 0,C 180,E1 29507.951,E2 29507.951} C_VEL
LIN {X 0,Y 632.895,Z 206.388,A -85,B 0,C 180,E1 29504.796,E2 29504.796} C_VEL
LIN {X 0,Y 632.858,Z 206.394,A -85,B 0,C 180,E1 29501.675,E2 29501.675} C_VEL
LIN {X 0,Y 632.894,Z 206.391,A -85,B 0,C 180,E1 29498.595,E2 29498.595} C_VEL
LIN {X 0,Y 632.851,Z 206.397,A -85,B 0,C 180,E1 29495.515,E2 29495.515} C_VEL
LIN {X 0,Y 632.893,Z 206.391,A -85,B 0,C 180,E1 29492.413,E2 29492.413} C_VEL
LIN {X 0,Y 632.847,Z 206.398,A -85,B 0,C 180,E1 29489.419,E2 29489.419} C_VEL
LIN {X 0,Y 632.894,Z 206.393,A -85,B 0,C 180,E1 29486.321,E2 29486.321} C_VEL
LIN {X 0,Y 632.842,Z 206.399,A -85,B 0,C 180,E1 29483.327,E2 29483.327} C_VEL
LIN {X 0,Y 632.896,Z 206.392,A -85,B 0,C 180,E1 29480.3,E2 29480.3} C_VEL
LIN {X 0,Y 632.838,Z 206.402,A -85,B 0,C 180,E1 29477.282,E2 29477.282} C_VEL
LIN {X 0,Y 632.9,Z 206.535,A -85,B 0,C 180,E1 29475.958,E2 29475.958} C_VEL
LIN {X 0,Y 633.936,Z 209.536,A -85,B 0,C 180,E1 29475.674,E2 29475.674} C_VEL
LIN {X 0,Y 635.232,Z 211.906,A -85,B 0,C 180,E1 29475.41,E2 29475.41} C_VEL
LIN {X 0,Y 645.759,Z 232.745,A -85,B 0,C 180,E1 29473.237,E2 29473.237} C_VEL
LIN {X 0,Y 653.974,Z 250.328,A -85,B 0,C 180,E1 29471.572,E2 29471.572} C_VEL
LIN {X 0,Y 651.046,Z 303.925,A -85,B 0,C 180,E1 29468.809,E2 29468.809} C_VEL
LIN {X 0,Y 653.477,Z 321.86,A -85,B 0,C 180,E1 29468.406,E2 29468.406} C_VEL
LIN {X 0,Y 650.878,Z 527.556,A -85,B 0,C 180,E1 29465.841,E2 29465.841} C_VEL
LIN {X 0,Y 648.936,Z 692.545,A -85,B 0,C 180,E1 29463.816,E2 29463.816} C_VEL
LIN {X 0,Y 648.205,Z 717.768,A -85,B 0,C 180,E1 29463.352,E2 29463.352} C_VEL
LIN {X 0,Y 647.368,Z 739.572,A -85,B 0,C 180,E1 29462.816,E2 29462.816} C_VEL
LIN {X 0,Y 646.169,Z 765.275,A -85,B 0,C 180,E1 29462.007,E2 29462.007} C_VEL
LIN {X 0,Y 645.045,Z 786.711,A -85,B 0,C 180,E1 29461.181,E2 29461.181} C_VEL
LIN {X 0,Y 643.662,Z 810.452,A -85,B 0,C 180,E1 29460.086,E2 29460.086} C_VEL
LIN {X 0,Y 642.593,Z 827.04,A -85,B 0,C 180,E1 29459.199,E2 29459.199} C_VEL
LIN {X 0,Y 641.236,Z 844.718,A -85,B 0,C 180,E1 29458.094,E2 29458.094} C_VEL
LIN {X 0,Y 639.571,Z 865.996,A -85,B 0,C 180,E1 29456.559,E2 29456.559} C_VEL
LIN {X 0,Y 638.241,Z 882.84,A -85,B 0,C 180,E1 29455.172,E2 29455.172} C_VEL
LIN {X 0,Y 636.789,Z 901.674,A -85,B 0,C 180,E1 29453.407,E2 29453.407} C_VEL
LIN {X 0,Y 635.682,Z 916.781,A -85,B 0,C 180,E1 29451.79,E2 29451.79} C_VEL
LIN {X 0,Y 634.573,Z 933.116,A -85,B 0,C 180,E1 29449.802,E2 29449.802} C_VEL
LIN {X 0,Y 633.767,Z 945.881,A -85,B 0,C 180,E1 29448.013,E2 29448.013} C_VEL
LIN {X 0,Y 633.093,Z 958.731,A -85,B 0,C 180,E1 29445.951,E2 29445.951} C_VEL
LIN {X 0,Y 632.626,Z 969.101,A -85,B 0,C 180,E1 29443.994,E2 29443.994} C_VEL
LIN {X 0,Y 632.302,Z 978.77,A -85,B 0,C 180,E1 29441.863,E2 29441.863} C_VEL
LIN {X 0,Y 632.087,Z 986.211,A -85,B 0,C 180,E1 29439.837,E2 29439.837} C_VEL
LIN {X 0,Y 631.97,Z 991.999,A -85,B 0,C 180,E1 29437.912,E2 29437.912} C_VEL
LIN {X 0,Y 631.917,Z 997.176,A -85,B 0,C 180,E1 29435.63,E2 29435.63} C_VEL
LIN {X 0,Y 631.915,Z 1000.124,A -85,B 0,C 180,E1 29433.72,E2 29433.72} C_VEL
LIN {X 0,Y 631.899,Z 1002.103,A -85,B 0,C 180,E1 29431.541,E2 29431.541} C_VEL
LIN {X 0,Y 631.884,Z 1002.373,A -85,B 0,C 180,E1 29429.456,E2 29429.456} C_VEL
LIN {X 0,Y 631.901,Z 1001.428,A -85,B 0,C 180,E1 29427.551,E2 29427.551} C_VEL
LIN {X 0,Y 631.914,Z 998.768,A -85,B 0,C 180,E1 29425.28,E2 29425.28} C_VEL
LIN {X 0,Y 631.945,Z 994.895,A -85,B 0,C 180,E1 29423.276,E2 29423.276} C_VEL
LIN {X 0,Y 632.003,Z 989.71,A -85,B 0,C 180,E1 29421.264,E2 29421.264} C_VEL
LIN {X 0,Y 632.177,Z 982.308,A -85,B 0,C 180,E1 29419.059,E2 29419.059} C_VEL
LIN {X 0,Y 632.428,Z 974.751,A -85,B 0,C 180,E1 29417.212,E2 29417.212} C_VEL
LIN {X 0,Y 632.849,Z 964.405,A -85,B 0,C 180,E1 29415.076,E2 29415.076} C_VEL
LIN {X 0,Y 633.384,Z 953.117,A -85,B 0,C 180,E1 29413.114,E2 29413.114} C_VEL
LIN {X 0,Y 634.153,Z 939.764,A -85,B 0,C 180,E1 29411.093,E2 29411.093} C_VEL
LIN {X 0,Y 635.062,Z 925.617,A -85,B 0,C 180,E1 29409.252,E2 29409.252} C_VEL
LIN {X 0,Y 636.186,Z 909.998,A -85,B 0,C 180,E1 29407.45,E2 29407.45} C_VEL
LIN {X 0,Y 637.46,Z 892.822,A -85,B 0,C 180,E1 29405.735,E2 29405.735} C_VEL
LIN {X 0,Y 638.907,Z 874.495,A -85,B 0,C 180,E1 29404.111,E2 29404.111} C_VEL
LIN {X 0,Y 640.439,Z 855.057,A -85,B 0,C 180,E1 29402.626,E2 29402.626} C_VEL
LIN {X 0,Y 642.047,Z 834.746,A -85,B 0,C 180,E1 29401.258,E2 29401.258} C_VEL
LIN {X 0,Y 643.264,Z 816.477,A -85,B 0,C 180,E1 29400.223,E2 29400.223} C_VEL
LIN {X 0,Y 644.351,Z 796.553,A -85,B 0,C 180,E1 29399.282,E2 29399.282} C_VEL
LIN {X 0,Y 645.536,Z 772.741,A -85,B 0,C 180,E1 29398.326,E2 29398.326} C_VEL
LIN {X 0,Y 646.466,Z 750.59,A -85,B 0,C 180,E1 29397.598,E2 29397.598} C_VEL
LIN {X 0,Y 647.321,Z 725.958,A -85,B 0,C 180,E1 29396.944,E2 29396.944} C_VEL
LIN {X 0,Y 647.966,Z 701.892,A -85,B 0,C 180,E1 29396.472,E2 29396.472} C_VEL
LIN {X 0,Y 648.405,Z 672.909,A -85,B 0,C 180,E1 29396.081,E2 29396.081} C_VEL
LIN {X 0,Y 649.549,Z 453.207,A -85,B 0,C 180,E1 29393.592,E2 29393.592} C_VEL
LIN {X 0,Y 650.483,Z 318.941,A -85,B 0,C 180,E1 29391.975,E2 29391.975} C_VEL
LIN {X 0,Y 649.032,Z 309.647,A -85,B 0,C 180,E1 29391.762,E2 29391.762} C_VEL
LIN {X 0,Y 651.379,Z 277.525,A -85,B 0,C 180,E1 29389.995,E2 29389.995} C_VEL
LIN {X 0,Y 654.506,Z 251.306,A -85,B 0,C 180,E1 29388.411,E2 29388.411} C_VEL
LIN {X 0,Y 652.582,Z 245.471,A -85,B 0,C 180,E1 29387.729,E2 29387.729} C_VEL
LIN {X 0,Y 649.431,Z 237.865,A -85,B 0,C 180,E1 29386.612,E2 29386.612} C_VEL
LIN {X 0,Y 646.808,Z 231.657,A -85,B 0,C 180,E1 29385.451,E2 29385.451} C_VEL
LIN {X 0,Y 644.659,Z 227.282,A -85,B 0,C 180,E1 29384.264,E2 29384.264} C_VEL
LIN {X 0,Y 643.167,Z 224.433,A -85,B 0,C 180,E1 29382.917,E2 29382.917} C_VEL
LIN {X 0,Y 643.014,Z 223.304,A -85,B 0,C 180,E1 29381.844,E2 29381.844} C_VEL
LIN {X 0,Y 642.996,Z 224.118,A -85,B 0,C 180,E1 29380.895,E2 29380.895} C_VEL
LIN {X 0,Y 644.221,Z 226.82,A -85,B 0,C 180,E1 29379.521,E2 29379.521} C_VEL
LIN {X 0,Y 644.754,Z 227.969,A -85,B 0,C 180,E1 29379.137,E2 29379.137} C_VEL
LIN {X 0,Y 646.517,Z 232.246,A -85,B 0,C 180,E1 29378.074,E2 29378.074} C_VEL
LIN {X 0,Y 648.723,Z 237.823,A -85,B 0,C 180,E1 29377.022,E2 29377.022} C_VEL
LIN {X 0,Y 651.64,Z 246.685,A -85,B 0,C 180,E1 29375.737,E2 29375.737} C_VEL
LIN {X 0,Y 648.257,Z 273.291,A -85,B 0,C 180,E1 29373.76,E2 29373.76} C_VEL
LIN {X 0,Y 644.469,Z 314.816,A -85,B 0,C 180,E1 29370.9,E2 29370.9} C_VEL
LIN {X 0,Y 641.686,Z 361.357,A -85,B 0,C 180,E1 29367.87,E2 29367.87} C_VEL
LIN {X 0,Y 639.385,Z 412.532,A -85,B 0,C 180,E1 29364.68,E2 29364.68} C_VEL
LIN {X 0,Y 638.327,Z 443.948,A -85,B 0,C 180,E1 29362.796,E2 29362.796} C_VEL
LIN {X 0,Y 642.421,Z 479.638,A -85,B 0,C 180,E1 29361.896,E2 29361.896} C_VEL
LIN {X 0,Y 642.916,Z 487.294,A -85,B 0,C 180,E1 29361.734,E2 29361.734} C_VEL
LIN {X 0,Y 639.482,Z 602.556,A -85,B 0,C 180,E1 29359.959,E2 29359.959} C_VEL
LIN {X 0,Y 637.883,Z 684.332,A -85,B 0,C 180,E1 29358.76,E2 29358.76} C_VEL
LIN {X 0,Y 637.375,Z 705.209,A -85,B 0,C 180,E1 29358.28,E2 29358.28} C_VEL
LIN {X 0,Y 636.827,Z 725.235,A -85,B 0,C 180,E1 29357.64,E2 29357.64} C_VEL
LIN {X 0,Y 636.236,Z 743.839,A -85,B 0,C 180,E1 29356.87,E2 29356.87} C_VEL
LIN {X 0,Y 635.678,Z 761.117,A -85,B 0,C 180,E1 29355.978,E2 29355.978} C_VEL
LIN {X 0,Y 635.104,Z 777.203,A -85,B 0,C 180,E1 29354.963,E2 29354.963} C_VEL
LIN {X 0,Y 634.553,Z 791.727,A -85,B 0,C 180,E1 29353.858,E2 29353.858} C_VEL
LIN {X 0,Y 634.047,Z 804.854,A -85,B 0,C 180,E1 29352.662,E2 29352.662} C_VEL
LIN {X 0,Y 633.605,Z 816.656,A -85,B 0,C 180,E1 29351.377,E2 29351.377} C_VEL
LIN {X 0,Y 633.221,Z 827.13,A -85,B 0,C 180,E1 29350.003,E2 29350.003} C_VEL
LIN {X 0,Y 632.901,Z 836.416,A -85,B 0,C 180,E1 29348.51,E2 29348.51} C_VEL
LIN {X 0,Y 632.672,Z 843.948,A -85,B 0,C 180,E1 29346.99,E2 29346.99} C_VEL
LIN {X 0,Y 632.518,Z 850.147,A -85,B 0,C 180,E1 29345.352,E2 29345.352} C_VEL
LIN {X 0,Y 632.398,Z 854.536,A -85,B 0,C 180,E1 29343.717,E2 29343.717} C_VEL
LIN {X 0,Y 632.326,Z 857.346,A -85,B 0,C 180,E1 29341.994,E2 29341.994} C_VEL
LIN {X 0,Y 632.291,Z 858.371,A -85,B 0,C 180,E1 29340.272,E2 29340.272} C_VEL
LIN {X 0,Y 632.271,Z 857.643,A -85,B 0,C 180,E1 29338.55,E2 29338.55} C_VEL
LIN {X 0,Y 632.288,Z 855.157,A -85,B 0,C 180,E1 29336.827,E2 29336.827} C_VEL
LIN {X 0,Y 632.334,Z 851.122,A -85,B 0,C 180,E1 29335.193,E2 29335.193} C_VEL
LIN {X 0,Y 632.435,Z 845.351,A -85,B 0,C 180,E1 29333.555,E2 29333.555} C_VEL
LIN {X 0,Y 632.606,Z 837.68,A -85,B 0,C 180,E1 29331.913,E2 29331.913} C_VEL
LIN {X 0,Y 632.877,Z 828.445,A -85,B 0,C 180,E1 29330.356,E2 29330.356} C_VEL
LIN {X 0,Y 633.234,Z 817.757,A -85,B 0,C 180,E1 29328.893,E2 29328.893} C_VEL
LIN {X 0,Y 633.675,Z 805.564,A -85,B 0,C 180,E1 29327.515,E2 29327.515} C_VEL
LIN {X 0,Y 634.214,Z 791.659,A -85,B 0,C 180,E1 29326.21,E2 29326.21} C_VEL
LIN {X 0,Y 634.805,Z 776.472,A -85,B 0,C 180,E1 29325.03,E2 29325.03} C_VEL
LIN {X 0,Y 635.425,Z 759.895,A -85,B 0,C 180,E1 29323.969,E2 29323.969} C_VEL
LIN {X 0,Y 636.005,Z 743.177,A -85,B 0,C 180,E1 29323.091,E2 29323.091} C_VEL
LIN {X 0,Y 636.595,Z 725.725,A -85,B 0,C 180,E1 29322.353,E2 29322.353} C_VEL
LIN {X 0,Y 637.118,Z 706.586,A -85,B 0,C 180,E1 29321.727,E2 29321.727} C_VEL
LIN {X 0,Y 637.572,Z 687.079,A -85,B 0,C 180,E1 29321.267,E2 29321.267} C_VEL
LIN {X 0,Y 637.92,Z 664.257,A -85,B 0,C 180,E1 29320.924,E2 29320.924} C_VEL
LIN {X 0,Y 640.189,Z 482.959,A -85,B 0,C 180,E1 29318.602,E2 29318.602} C_VEL
LIN {X 0,Y 637.648,Z 461.325,A -85,B 0,C 180,E1 29318.183,E2 29318.183} C_VEL
LIN {X 0,Y 638.723,Z 425.411,A -85,B 0,C 180,E1 29316.058,E2 29316.058} C_VEL
LIN {X 0,Y 638.011,Z 419.163,A -85,B 0,C 180,E1 29315.65,E2 29315.65} C_VEL
LIN {X 0,Y 632.689,Z 403.351,A -85,B 0,C 180,E1 29314.46,E2 29314.46} C_VEL
LIN {X 0,Y 632.169,Z 397.972,A -85,B 0,C 180,E1 29314.106,E2 29314.106} C_VEL
LIN {X 0,Y 634.213,Z 344.412,A -85,B 0,C 180,E1 29310.845,E2 29310.845} C_VEL
LIN {X 0,Y 636.346,Z 292.016,A -85,B 0,C 180,E1 29307.601,E2 29307.601} C_VEL
LIN {X 0,Y 638.577,Z 243.118,A -85,B 0,C 180,E1 29304.526,E2 29304.526} C_VEL
LIN {X 0,Y 628.677,Z 217.087,A -85,B 0,C 180,E1 29302.154,E2 29302.154} C_VEL
LIN {X 0,Y 624.895,Z 207.391,A -85,B 0,C 180,E1 29301.226,E2 29301.226} C_VEL
LIN {X 0,Y 624.9,Z 207.391,A -85,B 0,C 180,E1 29297.899,E2 29297.899} C_VEL
LIN {X 0,Y 624.949,Z 207.381,A -85,B 0,C 180,E1 29294.864,E2 29294.864} C_VEL
LIN {X 0,Y 624.933,Z 207.387,A -85,B 0,C 180,E1 29291.651,E2 29291.651} C_VEL
LIN {X 0,Y 624.928,Z 207.584,A -85,B 0,C 180,E1 29289.737,E2 29289.737} C_VEL
LIN {X 0,Y 626.015,Z 210.6,A -85,B 0,C 180,E1 29289.472,E2 29289.472} C_VEL
LIN {X 0,Y 632.721,Z 226.25,A -85,B 0,C 180,E1 29287.947,E2 29287.947} C_VEL
LIN {X 0,Y 640.273,Z 245.58,A -85,B 0,C 180,E1 29286.007,E2 29286.007} C_VEL
LIN {X 0,Y 640.705,Z 247.691,A -85,B 0,C 180,E1 29285.819,E2 29285.819} C_VEL
LIN {X 0,Y 639.221,Z 289.191,A -85,B 0,C 180,E1 29282.767,E2 29282.767} C_VEL
LIN {X 0,Y 638.897,Z 318.308,A -85,B 0,C 180,E1 29280.773,E2 29280.773} C_VEL
LIN {X 0,Y 639.099,Z 324.989,A -85,B 0,C 180,E1 29280.363,E2 29280.363} C_VEL
LIN {X 0,Y 639.536,Z 329.306,A -85,B 0,C 180,E1 29280.282,E2 29280.282} C_VEL
LIN {X 0,Y 637.723,Z 440.539,A -85,B 0,C 180,E1 29278.862,E2 29278.862} C_VEL
LIN {X 0,Y 634.236,Z 617.38,A -85,B 0,C 180,E1 29276.398,E2 29276.398} C_VEL
LIN {X 0,Y 633.701,Z 640.001,A -85,B 0,C 180,E1 29275.917,E2 29275.917} C_VEL
LIN {X 0,Y 632.964,Z 662.226,A -85,B 0,C 180,E1 29275.272,E2 29275.272} C_VEL
LIN {X 0,Y 632.12,Z 684.246,A -85,B 0,C 180,E1 29274.449,E2 29274.449} C_VEL
LIN {X 0,Y 631.255,Z 703.32,A -85,B 0,C 180,E1 29273.575,E2 29273.575} C_VEL
LIN {X 0,Y 630.24,Z 722.986,A -85,B 0,C 180,E1 29272.48,E2 29272.48} C_VEL
